I120_REJ_BIN_PRSNCE_I1221_0                    :BOOL;
I120_SPARE_I1221_1                             :BOOL;
I120_SPARE_I1221_2                             :BOOL;
I120_SPARE_I1221_3                             :BOOL;
I120_SPARE_I1221_4                             :BOOL;
I120_SPARE_I1221_5                             :BOOL;
I120_SPARE_I1221_6                             :BOOL;
I120_SPARE_I1221_7                             :BOOL;

//port 5
O90_RET_LH_GRIPR_CYL_CLSE_Q1240_0              :BOOL;
O90_RET_LH_GRIPR_CYL_OPN_Q1240_1               :BOOL;
O90_RET_RH_GRIPR_CYL_CLSE_Q1240_2              :BOOL;
O90_RET_RH_GRIPR_CYL_OPN_Q1240_3               :BOOL;
O90_POS_LOCK_CYL1_VLVE_1_Q1240_4               :BOOL;
O90_POS_LOCK_CYL1_VLVE_2_Q1240_5               :BOOL;
O90_POS_LOCK_CYL2_VLVE_1_Q1240_6               :BOOL;
O90_POS_LOCK_CYL2_VLVE_2_Q1240_7               :BOOL;
											  
O90_POSTN_SLIDE_CYL_REV_Q1241_0                :BOOL;
O90_POSTN_SLIDE_CYL_FWD_Q1241_1                :BOOL;
O90_LH_MOVR_SUP_VERT_CYL_DWN_Q1241_2           :BOOL;
O90_LH_MOVR_SUP_VERT_CYL_UP_Q1241_3            :BOOL;
O90_LH_MOVR_SUP_HORZ_CYL_REV_Q1241_4           :BOOL;
O90_LH_MOVR_SUP_HORZ_CYL_FWD_Q1241_5           :BOOL;
O90_RH_MOVR_SUP_VERT_CYL_DWN_Q1241_6           :BOOL;
O90_RH_MOVR_SUP_VERT_CYL_UP_Q1241_7            :BOOL;
											   
O90_RH_MOVR_SUP_HORZ_CYL_REV_Q1242_0           :BOOL;
O90_RH_MOVR_SUP_HORZ_CYL_FWD_Q1242_1           :BOOL;
O90_SPARE_Q1242_2                              :BOOL;
O90_SPARE_Q1242_3                              :BOOL;
O90_SPARE_Q1242_4                              :BOOL;
O90_SPARE_Q1242_5                              :BOOL;
O90_SPARE_Q1242_6                              :BOOL;
O90_SPARE_Q1242_7                              :BOOL;

//port6
O90_LH1_REJ_SLIDE_REV_Q1250_0                  :BOOL;
O90_LH1_REJ_SLIDE_FWD_Q1250_1                  :BOOL;
O90_RH1_REJ_SLIDE_REV_Q1250_2                  :BOOL;
O90_RH1_REJ_SLIDE_FWD_Q1250_3                  :BOOL;
O90_SPARE_Q1250_4                              :BOOL;
O90_LH1_REJ_AIR_PURGE_Q1250_5                  :BOOL;
O90_LH2_REJ_SLIDE_REV_Q1250_6                  :BOOL;
O90_LH2_REJ_SLIDE_FWD_Q1250_7                  :BOOL;
											  
O90_RH2_REJ_SLIDE_REV_Q1251_0                  :BOOL;
O90_RH2_REJ_SLIDE_FWD_Q1251_1                  :BOOL;
O90_RH_REJ_AIR_PURGE_Q1251_2                   :BOOL;
O90_SPARE_Q1251_3                              :BOOL;
O90_SPARE_Q1251_4                              :BOOL;
O90_SPARE_Q1251_5                              :BOOL;
O90_SPARE_Q1251_6                              :BOOL;
O90_SPARE_Q1251_7                              :BOOL;

//port7
O110_LH_OIL_DISPN_ON_Q1260_0                   :BOOL;
O110_LH_OIL_SPIN_ON_Q1260_1                    :BOOL;
O110_RH_OIL_DISPN_ON_Q1260_2                   :BOOL;
O110_RH_OIL_SPIN_ON_Q1260_3                    :BOOL;
O120_LH_GRPR_CLSE_Q1260_4                      :BOOL;
O120_LH_GRPR_OPN_Q1260_5                       :BOOL;
O120_RH_GRPR_CLSE_Q1260_6                      :BOOL;
O120_RH_GRPR_OPN_Q1260_7                       :BOOL;
											  
O120_TOOL_CHO_UNLOCK_Q1261_0                   :BOOL;
O120_TOOL_CHO_LOCK_Q1261_1                     :BOOL;
O120_PUSH_CYL_REV_Q1261_2                      :BOOL;
O120_PUSH_CYL_FWD_Q1261_3                      :BOOL;
O120_LH_SING_CYL_REV_Q1261_4                   :BOOL;
O120_LH_SING_CYL_FWD_Q1261_5                   :BOOL;
O120_LH_REJ_AIR_PURGE_Q1261_6                  :BOOL;
O120_RH_REJ_AIR_PURGE_Q1261_7                  :BOOL;
											  
O120_CAMERA_SLIDECYL_REV_Q1262_0               :BOOL;
O120_CAMERA_SLIDECYL_FWD_Q1262_1               :BOOL;
O120_SPARE_Q1262_2                             :BOOL;
O120_SPARE_Q1262_3                             :BOOL;
O120_SPARE_Q1262_4                             :BOOL;
O120_SPARE_Q1262_5                             :BOOL;
O120_SPARE_Q1262_6                             :BOOL;
O120_SPARE_Q1262_7                             :BOOL;
END_VAR

// ---- POUs/IO_GVLs/Master4_IO.TcGVL

VAR_GLOBAL
//port1					
I130_LH_ROTRY_0_DEGI1300_0                :BOOL;
I130_LH_ROTRY_180_DEGI1300_1              :BOOL;
I130_RH_ROTRY_0_DEGI1300_2                :BOOL;
I130_RH_ROTRY_180_DEGI1300_3              :BOOL;
I130_SPARE_I1300_4                        :BOOL;
I130_SPARE_I1300_5                        :BOOL;
I130_SPARE_I1300_6                        :BOOL;
I130_SPARE_I1300_7                        :BOOL;
										  
I140_HORZ_SUP1_CYL_REVI1301_0             :BOOL;
I140_HORZ_SUP1_CYL_FWDI1301_1             :BOOL;
I140_VERT_SUP1_CYL_REVI1301_2             :BOOL;
I140_VERT_SUP1_CYL_FWDI1301_3             :BOOL;
I140_WIPE1_CYL_REVI1301_4                 :BOOL;
I140_WIPE1_CYL_FWDI1301_5                 :BOOL;
I140_SPARE_I1301_6                        :BOOL;
I140_SPARE_I1301_7                        :BOOL;
										  
// port 2                         
I140_HORZ_SUP2_CYL_REVI1310_0             :BOOL;
I140_HORZ_SUP2_CYL_FWDI1310_1             :BOOL;
I140_VERT_SUP2_CYL_REVI1310_2             :BOOL;
I140_VERT_SUP2_CYL_FWDI1310_3             :BOOL;
I140_WIPE2_CYL_REVI1310_4                 :BOOL;
I140_WIPE2_CYL_FWDI1310_5                 :BOOL;
I140_HORZ_SUP3_CYL_REVI1310_6             :BOOL;
I140_HORZ_SUP3_CYL_FWDI1310_7             :BOOL;
										  
I140_VERT_SUP3_CYL_REVI1311_0             :BOOL;
I140_VERT_SUP3_CYL_FWDI1311_1             :BOOL;
I140_WIPE3_CYL_REVI1311_2                 :BOOL;
I140_WIPE3_CYL_FWDI1311_3                 :BOOL;
I140_LEAKTEST_PRESS_SWI1311_4             :BOOL;
I140_SPARE_I1311_5                        :BOOL;
I160_MOVR_REM_CYL_REVI1311_6             :BOOL;
I160_MOVR_REM_CYL_FWDI1311_7             :BOOL;
										  
// port 3                        									  
I160_SLIDE_CYL_REVI1320_0                 :BOOL;
I160_SLIDE_CYL_FWDI1320_1                 :BOOL;
I160_SLAVE1_PRSN_PARK_TRAYI1320_2         :BOOL;
I160_SLAVE2_PRSN_PARK_TRAYI1320_3         :BOOL;
I160_FIXT_COMP1_PRSNI1320_4               :BOOL;
I160_FIXT_COMP2_PRSNI1320_5               :BOOL;
I160_SPARE_I1320_6                        :BOOL;
I160_SPARE_I1320_7                        :BOOL;
										  
I160_SPARE_I1321_0                        :BOOL;
I160_SPARE_I1321_1                        :BOOL;
I160_SPARE_I1321_2                        :BOOL;
I160_SPARE_I1321_3                        :BOOL;
I160_SPARE_I1321_4                        :BOOL;
I160_SPARE_I1321_5                        :BOOL;
I160_SPARE_I1321_6                        :BOOL;
I160_SPARE_I1321_7                        :BOOL;
										  
// port 4                        
I160_LH_PALLET_LOCK_CYL_UNLOCKI1330_0     :BOOL;
I160_LH_PALLET_LOCK_CYL_LOCKI1330_1       :BOOL;
I160_RH_PALLET_LOCK_CYL_UNLOCKI1330_2     :BOOL;
I160_RH_PALLET_LOCK_CYL_LOCKI1330_3       :BOOL;
I160_SPARE_I1330_4                        :BOOL;
I160_CONV_BDY_PRSN1_SENI1330_5            :BOOL;
I160_CONV_BDY_PRSN2_SENI1330_6            :BOOL;
I160_SPARE_I1330_7                        :BOOL;
										  
I160_REJ_BOX_DOOR_CLSEI1331_0             :BOOL;
I160_SAM_PART_BAG_DOOR_CLSEI1331_1        :BOOL;
I160_TROLLEY_FIXT_PRSNI1331_2             :BOOL;
I160_SAM_BOX_DOOR_CLSEI1331_3             :BOOL;
I160_SPARE_I1331_4                        :BOOL;
I160_SPARE_I1331_5                        :BOOL;
I160_SPARE_I1331_6                        :BOOL;
I160_SPARE_I1331_7                        :BOOL;
										 
//PORT5                            									 
O130_LH_ROTRY_0_DEG_Q1340_0               :BOOL;
O130_LH_ROTRY_180_DEG_Q1340_1             :BOOL;
O130_RH_ROTRY_0_DEG_Q1340_2               :BOOL;
O130_RH_ROTRY_180_DEG_Q1340_3             :BOOL;
O130_LH_TOOL_CHO_UNLOCK_Q1340_4           :BOOL;
O130_LH_TOOL_CHO_LOCK_Q1340_5             :BOOL;
O130_RH_TOOL_CHO_UNLOCK_Q1340_6           :BOOL;
O130_RH_TOOL_CHO_LOCK_Q1340_7             :BOOL;
										 
O140_HORZ_SUP1_CYL_REV_Q1341_0            :BOOL;
O140_HORZ_SUP1_CYL_FWD_Q1341_1            :BOOL;
O140_VERT_SUP1_CYL_REV_Q1341_2            :BOOL;
O140_VERT_SUP1_CYL_FWD_Q1341_3            :BOOL;
O140_TOOL1_CHO_UNLOCK_Q1341_4             :BOOL;
O140_TOOL1_CHO_LOCK_Q1341_5               :BOOL;
O140_WIPE1_CYL_REV_Q1341_6                :BOOL;
O140_WIPE1_CYL_FWD_Q1341_7                :BOOL;
										  
O140_HORZ_SUP2_CYL_REV_Q1342_0            :BOOL;
O140_HORZ_SUP2_CYL_FWD_Q1342_1            :BOOL;
O140_VERT_SUP2_CYL_REV_Q1342_2            :BOOL;
O140_VERT_SUP2_CYL_FWD_Q1342_3            :BOOL;
O140_TOOL2_CHO_UNLOCK_Q1342_4             :BOOL;
O140_TOOL2_CHO_LOCK_Q1342_5               :BOOL;
O140_WIPE2_CYL_REV_Q1342_6                :BOOL;
O140_WIPE2_CYL_FWD_Q1342_7                :BOOL;
										  
O140_HORZ_SUP3_CYL_REV_Q1343_0            :BOOL;
O140_HORZ_SUP3_CYL_FWD_Q1343_1            :BOOL;
O140_VERT_SUP3_CYL_REV_Q1343_2            :BOOL;
O140_VERT_SUP3_CYL_FWD_Q1343_3            :BOOL;
O140_TOOL3_CHO_UNLOCK_Q1343_4             :BOOL;
O140_TOOL3_CHO_LOCK_Q1343_5               :BOOL;
O140_WIPE3_CYL_REV_Q1343_6                :BOOL;
O140_WIPE3_CYL_FWD_Q1343_7                :BOOL;
										  
//PORT6                           									  
O160_VISN_CHECK_AIR_PURGE_Q1350_0         :BOOL;
O160_FIXT_PP_GRPR_CLSE_OPN_Q1350_1        :BOOL;
O160_LH_COMP_PP_GRPR_CLSE_OPN_Q1350_2     :BOOL;
O160_RH_COMP_PP_GRPR_CLSE_OPN_Q1350_3     :BOOL;
O160_SLIDE_CYL_REV_Q1350_4                :BOOL;
O160_SLIDE_CYL_FWD_Q1350_5                :BOOL;
O160_SPARE_Q1350_6                        :BOOL;
O160_SPARE_Q1350_7                        :BOOL;
										 
O160_TOOL_CHO_UNLOCK_Q1351_0              :BOOL;
O160_TOOL_CHO_LOCK_Q1351_1                :BOOL;
O160_LH_PALLET_LOCK_CYL_UNLOCK_Q1351_2    :BOOL;
O160_LH_PALLET_LOCK_CYL_LOCK_Q1351_3      :BOOL;
O160_RH_PALLET_LOCK_CYL_UNLOCK_Q1351_4    :BOOL;
O160_RH_PALLET_LOCK_CYL_LOCK_Q1351_5      :BOOL;
O160_SPARE_Q1351_6                        :BOOL;
O160_SPARE_Q1351_7                        :BOOL;
										  
O160_SPARE_Q1352_0                        :BOOL;
O160_SPARE_Q1352_1                        :BOOL;
OP160_MOVR_REM_CYL_REV_Q1352_2           :BOOL;
OP160_MOVR_REM_CYL_FWD_Q1352_3           :BOOL;
O160_SPARE_Q1352_4                        :BOOL;
O160_SPARE_Q1352_5                        :BOOL;
O160_SPARE_Q1352_6                        :BOOL;
O160_SPARE_Q1352_7                        :BOOL;
										 
O160_SPARE_Q1353_0                        :BOOL;
O160_SPARE_Q1353_1                        :BOOL;
O160_SPARE_Q1353_2                        :BOOL;
O160_SPARE_Q1353_3                        :BOOL;
O160_SPARE_Q1353_4                        :BOOL;
O160_SPARE_Q1353_5                        :BOOL;
O160_SPARE_Q1353_6                        :BOOL;
O160_SPARE_Q1353_7                        :BOOL;
END_VAR

// ---- POUs/IO_GVLs/OP120_JB.TcGVL

VAR_GLOBAL

I120_SPARE_600_0I600_0             :BOOL;
I120_HPR_LOW_LVL_FBI600_1          :BOOL;
I120_HPR_SOL_DOOR_SW_FBI600_2      :BOOL;
I120_BOWL_RDYI600_3                :BOOL;
I120_BOWL_LOW_LVLI600_4            :BOOL;
I120_BOWL_OFF_ONI600_5             :BOOL;
I120_HPR_OFF_ONI600_6              :BOOL;
I120_CONV_REVI600_7                :BOOL;
I120_CONV_FWDI601_0                :BOOL;
I120_VBF_CONV_TRK1_OVERFLW_I601_1  :BOOL;
I120_VBF_CONV_TRK2_OVERFLWI601_2   :BOOL;
I120_CONV_TRK1_CHO_MOD1I601_3      :BOOL;
I120_CONV_TRK1_CHO_MOD2I601_4      :BOOL;
I120_CONV_TRK2_CHO_MOD1I601_5      :BOOL;
I120_CONV_TRK2_CHO_MOD2I601_6      :BOOL;
I120_CONV_TRK3_CHO_MOD1I601_7      :BOOL;
								   			   
I120_CONV_TRK3_CHO_MOD2I602_0      :BOOL;
I120_VBF_CONV_TRK_OVERFLW2_I602_1  :BOOL;
I120_SPARE_I602_2                  :BOOL;
I120_SPARE_I602_3                  :BOOL;
I120_SPARE_I602_4                  :BOOL;
I120_SPARE_I602_5                  :BOOL;
I120_SPARE_I602_6                  :BOOL;
I120_SPARE_I602_7                  :BOOL;
I120_SPARE_I603_0                  :BOOL;
I120_SPARE_I603_1                  :BOOL;
I120_SPARE_I603_2                  :BOOL;
I120_SPARE_I603_3                  :BOOL;
I120_SPARE_I603_4                  :BOOL;
I120_SPARE_I603_5                  :BOOL;
I120_SPARE_I603_6                  :BOOL;
I120_SPARE_I603_7                  :BOOL;

O120_HPR_ENABLEQ600_0              :BOOL;
O120_BOWL_ENABLEQ600_1             :BOOL;
O120_HPR_TWR_LMP_REDQ600_2         :BOOL;
O120_HPR_TWR_LMP_GREENQ600_3       :BOOL;
O120_BOWL_AIR_PURGE1Q600_4         :BOOL;
O120_BOWL_AIR_PURGE2Q600_5         :BOOL;
O120_HPR_DOOR_OPNQ600_6            :BOOL;
O120_SPARE_Q600_7                  :BOOL;
O120_SPARE_Q601_0                  :BOOL;
O120_SPARE_Q601_1                  :BOOL;
O120_SPARE_Q601_2                  :BOOL;
O120_SPARE_Q601_3                  :BOOL;
O120_SPARE_Q601_4                  :BOOL;
O120_SPARE_Q601_5                  :BOOL;
O120_SPARE_Q601_6                  :BOOL;
O120_SPARE_Q601_7                  :BOOL;

O120_SPARE_Q602_0                  :BOOL;
O120_SPARE_Q602_1                  :BOOL;
O120_SPARE_Q602_2                  :BOOL;
O120_SPARE_Q602_3                  :BOOL;
O120_SPARE_Q602_4                  :BOOL;
O120_SPARE_Q602_5                  :BOOL;
O120_SPARE_Q602_6                  :BOOL;
O120_SPARE_Q602_7                  :BOOL;
O120_SPARE_Q603_0                  :BOOL;
O120_SPARE_Q603_1                  :BOOL;
O120_SPARE_Q603_2                  :BOOL;
O120_SPARE_Q603_3                  :BOOL;
O120_SPARE_Q603_4                  :BOOL;
O120_SPARE_Q603_5                  :BOOL;
O120_SPARE_Q603_6                  :BOOL;
O120_SPARE_Q603_7                  :BOOL;
	
END_VAR

// ---- POUs/IO_GVLs/OP160_MP.TcGVL

VAR_GLOBAL
I130_LH_ATC_DECLAMP_FBI700_0				:BOOL;
I130_LH_ATC_CLAMP_FBI700_1                 :BOOL;
I130_LH_ATC_STN_POKE_YOKE_1I700_2          :BOOL;
I130_LH_ATC_STN_POKE_YOKE_2I700_3          :BOOL;
I130_LH_ATC_STN_POKE_YOKE_3I700_4          :BOOL;
I130_LH_ATC_STN_POKE_YOKE_4I700_5          :BOOL;
I130_LH_ATC_SLAVE_MODL1I700_6              :BOOL;
I130_LH_ATC_SLAVE_MODL2I700_7              :BOOL;
I130_RH_ATC_DECLAMP_FBI701_0               :BOOL;
I130_RH_ATC_CLAMP_FBI701_1                 :BOOL;
I130_RH_ATC_STN_POKE_YOKE_1I701_2          :BOOL;
I130_RH_ATC_STN_POKE_YOKE_2I701_3          :BOOL;
I130_RH_ATC_STN_POKE_YOKE_3I701_4          :BOOL;
I130_RH_ATC_STN_POKE_YOKE_4I701_5          :BOOL;
I130_RH_ATC_SLAVE_MODL1I701_6              :BOOL;
I130_RH_ATC_SLAVE_MODL2I701_7              :BOOL;

I140_ATC1_DECLAMP_FBI702_0                 :BOOL;
I140_ATC1_CLAMP_FBI702_1                   :BOOL;
I140_ATC1_STN_POKE_YOKE_1I702_2            :BOOL;
I140_ATC1_STN_POKE_YOKE_2I702_3            :BOOL;
I140_ATC1_STN_POKE_YOKE_3I702_4            :BOOL;
I140_ATC1_STN_POKE_YOKE_4I702_5            :BOOL;
I140_ATC1_SLAVE_MODL1I702_6                :BOOL;
I140_ATC1_SLAVE_MODL2I702_7                :BOOL;
I140_SPARE_I703_0                          :BOOL;
I140_SPARE_I703_1                          :BOOL;
I140_SPARE_I703_2                          :BOOL;
I140_LK_TST_1_PASI703_3                    :BOOL;
I140_LK_TST_1_FLI703_4                     :BOOL;
I140_LK_TST_1_REF_PRT_FLI703_5             :BOOL;
I140_LK_TST_1_WARNGI703_6                  :BOOL;
I140_LK_TST_1_END_CYCI703_7                :BOOL;

										  
I140_SPARE_I704_0I704_0                    :BOOL;
I140_LK_TST_2_PASI704_1                    :BOOL;
I140_LK_TST_2_FLI704_2                     :BOOL;
I140_LK_TST_2_REF_PRT_FLI704_3             :BOOL;
I140_LK_TST_2_WARNGI704_4                  :BOOL;
I140_LK_TST_2_END_CYCI704_5                :BOOL;
I140_SPARE_I704_6                          :BOOL;
I140_SPARE_I704_7                          :BOOL;
I140_ATC2_DECLAMP_FBI705_0                 :BOOL;
I140_ATC2_CLAMP_FBI705_1                   :BOOL;
I140_ATC2_STN_POKE_YOKE_1I705_2            :BOOL;
I140_ATC2_STN_POKE_YOKE_2I705_3            :BOOL;
I140_ATC2_STN_POKE_YOKE_3I705_4            :BOOL;
I140_ATC2_STN_POKE_YOKE_4I705_5            :BOOL;
I140_ATC2_SLAVE_MODL1I705_6                :BOOL;
I140_ATC2_SLAVE_MODL2I705_7                :BOOL;
										   

I140_SPARE_I706_0                          :BOOL;
I140_LK_TST_3_PASI706_1                    :BOOL;
I140_LK_TST_3_FLI706_2                     :BOOL;
I140_LK_TST_3_REF_PRT_FLI706_3             :BOOL;
I140_LK_TST_3_WARNGI706_4                  :BOOL;
I140_LK_TST_3_END_CYCI706_5                :BOOL;
I140_SPARE_I706_6                          :BOOL;
I140_SPARE_I706_7                          :BOOL;
I140_SPARE_I707_0                          :BOOL;
I140_LK_TST_4_PASI707_1                    :BOOL;
I140_LK_TST_4_FLI707_2                     :BOOL;
I140_LK_TST_4_REF_PRT_FLI707_3             :BOOL;
I140_LK_TST_4_WARNGI707_4                  :BOOL;
I140_LK_TST_4_END_CYCI707_5                :BOOL;
I140_SPARE_I707_6                          :BOOL;
I140_SPARE_I707_7                          :BOOL;


I140_ATC3_DECLAMP_FBI708_0                 :BOOL;
I140_ATC3_CLAMP_FBI708_1                   :BOOL;
I140_ATC3_STN_POKE_YOKE_1I708_2            :BOOL;
I140_ATC3_STN_POKE_YOKE_2I708_3            :BOOL;
I140_ATC3_STN_POKE_YOKE_3I708_4            :BOOL;
I140_ATC3_STN_POKE_YOKE_4I708_5            :BOOL;
I140_ATC3_SLAVE_MODL1I708_6                :BOOL;
I140_ATC3_SLAVE_MODL2I708_7                :BOOL;
I140_SPARE_I709_0                          :BOOL;
I140_SPARE_I709_1                          :BOOL;
I140_SPARE_I709_2                          :BOOL;
I140_LK_TST_5_PASI709_3                    :BOOL;
I140_LK_TST_5_FLI709_4                     :BOOL;
I140_LK_TST_5_REF_PRT_FLI709_5             :BOOL;
I140_LK_TST_5_WARNGI709_6                  :BOOL;
I140_LK_TST_5_END_CYCI709_7                :BOOL;

I140_SPARE_I710_0                          :BOOL;
I140_LK_TST_6_PASI710_1                    :BOOL;
I140_LK_TST_6_FLI710_2                     :BOOL;
I140_LK_TST_6_REF_PRT_FLI710_3             :BOOL;
I140_LK_TST_6_WARNGI710_4                  :BOOL;
I140_LK_TST_6_END_CYCI710_5                :BOOL;
I160_ATC_DECLAMP_FBI710_6                  :BOOL;
I160_ATC_CLAMP_FBI710_7                    :BOOL;
I160_ATC1_STN_POKE_YOKE_1I711_0            :BOOL;
I160_ATC1_STN_POKE_YOKE_2I711_1            :BOOL;
I160_ATC1_STN_POKE_YOKE_3I711_2            :BOOL;
I160_ATC1_STN_POKE_YOKE_4I711_3            :BOOL;
I160_ATC1_SLAVE_TOOL1I711_4                :BOOL;
I160_ATC1_SLAVE_TOOL2I711_5                :BOOL;
I160_FIXT_LH_COMP_PP_GRPR_CLSEI711_6       :BOOL;
I160_FIXT_LH_COMP_PP_GRPR_OPNI711_7        :BOOL;
I160_RH_COMP_PP_GRPR_CLSEI712_0            :BOOL;
I160_RH_COMP_PP_GRPR_OPNI712_1             :BOOL;
I160_AUTOBAG_READYI712_2                   :BOOL;
I160_SPARE_I712_3                          :BOOL;
I160_SPARE_I712_4                          :BOOL;
I160_AUTOBAG_ERR_STOPI712_5                :BOOL;
I20_RESRVR_LW_LVLI712_6                    :BOOL;
I20_OILTANK_PRES_SW_FBI712_7               :BOOL;
I160_SPARE_I713_0                          :BOOL;
I160_SPARE_I713_1                          :BOOL;
I160_VFD_RDYI713_2                         :BOOL;
I160_SPARE_I713_3                          :BOOL;
I160_SPARE_I713_4                          :BOOL;
I160_SPARE_I713_5                          :BOOL;
I160_SPARE_I713_6                          :BOOL;
I160_SPARE_I713_7                          :BOOL;


I10A_DRUM_FEED_ALRMI714_0                  :BOOL;
I10A_SPARE_I714_1                          :BOOL;
I10A_DRUM_OFF_ON_I714_2                    :BOOL;
I10A_DRUM_CONV_REV_I714_3                  :BOOL;
I10A_DRUM_CONV_FWD_I714_4                  :BOOL;
I10A_ROB_MAN_AUTO_MODE_I714_5              :BOOL;
I160_SPARE_I714_6                          :BOOL;
I160_SPARE_I714_7                          :BOOL;
I160_SPARE_I715_0                          :BOOL;
I160_SPARE_I715_1                          :BOOL;
I160_SPARE_I715_2                          :BOOL;
I160_SPARE_I715_3                          :BOOL;
I160_SPARE_I715_4                          :BOOL;
I160_SPARE_I715_5                          :BOOL;
I160_SPARE_I715_6                          :BOOL;
I160_SPARE_I715_7                          :BOOL;

O140_LK_TST1_RST_Q700_0                   :BOOL;
O140_LK_TST1_STRT_Q700_1                  :BOOL;
O140_LK_TST1_SEL1_Q700_2                  :BOOL;
O140_LK_TST1_SEL2_Q700_3                  :BOOL;
O140_LK_TST1_SEL3_Q700_4                  :BOOL;
O140_LK_TST1_SEL4_Q700_5                  :BOOL;
O140_LK_TST1_SEL5_Q700_6                  :BOOL;
O140_LK_TST1_SEL6_Q700_7                  :BOOL;
O140_LK_TST1_SEL7_Q701_0                  :BOOL;
O140_LK_TST2_RST_Q701_1                   :BOOL;
O140_LK_TST2_STRT_Q701_2                  :BOOL;
O140_LK_TST2_SEL1_Q701_3                  :BOOL;
O140_LK_TST2_SEL2_Q701_4                  :BOOL;
O140_LK_TST2_SEL3_Q701_5                  :BOOL;
O140_LK_TST2_SEL4_Q701_6                  :BOOL;
O140_LK_TST2_SEL5_Q701_7                  :BOOL;

O140_LK_TST2_SEL6_Q702_0                  :BOOL;
O140_LK_TST2_SEL7_Q702_1                  :BOOL;
O140_LK_TST3_RST_Q702_2                   :BOOL;
O140_LK_TST3_STRT_Q702_3                  :BOOL;
O140_LK_TST3_SEL1_Q702_4                  :BOOL;
O140_LK_TST3_SEL2_Q702_5                  :BOOL;
O140_LK_TST3_SEL3_Q702_6                  :BOOL;
O140_LK_TST3_SEL4_Q702_7                  :BOOL;
O140_LK_TST3_SEL5_Q703_0                  :BOOL;
O140_LK_TST3_SEL6_Q703_1                  :BOOL;
O140_LK_TST3_SEL7_Q703_2                  :BOOL;
O140_LK_TST4_RST_Q703_3                   :BOOL;
O140_LK_TST4_STRT_Q703_4                  :BOOL;
O140_LK_TST4_SEL1_Q703_5                  :BOOL;
O140_LK_TST4_SEL2_Q703_6                  :BOOL;
O140_LK_TST4_SEL3_Q703_7                  :BOOL;

O140_LK_TST4_SEL4_Q704_0                  :BOOL;
O140_LK_TST4_SEL5_Q704_1                  :BOOL;
O140_LK_TST4_SEL6_Q704_2                  :BOOL;
O140_LK_TST4_SEL7_Q704_3                  :BOOL;
O140_LK_TST5_RST_Q704_4                   :BOOL;
O140_LK_TST5_STRT_Q704_5                  :BOOL;
O140_LK_TST5_SEL1_Q704_6                  :BOOL;
O140_LK_TST5_SEL2_Q704_7                  :BOOL;
O140_LK_TST5_SEL3_Q705_0                  :BOOL;
O140_LK_TST5_SEL4_Q705_1                  :BOOL;
O140_LK_TST5_SEL5_Q705_2                  :BOOL;
O140_LK_TST5_SEL6_Q705_3                  :BOOL;
O140_LK_TST5_SEL7_Q705_4                  :BOOL;
O140_LK_TST6_RST_Q705_5                   :BOOL;
O140_LK_TST6_STRT_Q705_6                  :BOOL;
O140_LK_TST6_SEL1_Q705_7                  :BOOL;
										   

O140_LK_TST6_SEL2_Q706_0                  :BOOL;
O140_LK_TST6_SEL3_Q706_1                  :BOOL;
O140_LK_TST6_SEL4_Q706_2                  :BOOL;
O140_LK_TST6_SEL5_Q706_3                  :BOOL;
O140_LK_TST6_SEL6_Q706_4                  :BOOL;
O140_LK_TST6_SEL7_Q706_5                  :BOOL;
O150_VISN_LGHT_ON_Q706_6                   :BOOL;
O150_BARLIGHT_OP1_Q706_7                   :BOOL;
O150_BARLIGHT_OP2_Q707_0                   :BOOL;
O160_CHECKER_LGHT_ON_Q707_1                :BOOL;
O160_FUME_EXTRTR_ON_Q707_2                 :BOOL;
O160_MC_LMP_ON_Q707_3                      :BOOL;
O160_AUTOBAG_CNT_CMPLTD_Q707_4             :BOOL;
O160_SAMPLE_PART_DOOR_OPN_Q707_5           :BOOL;
O160_REJ_BIN_DOOR_OPN_Q707_6               :BOOL;
O160_SPARE_Q707_7                          :BOOL;
										   
O160_VFD_FWD_Q708_0                        :BOOL;
O160_VFD_REV_Q708_1                        :BOOL;
O160_VFD_STOP_Q708_2                       :BOOL;
O160_BOT_MC_LMP_ON_Q708_3                  :BOOL;
O10A_DRUM_MTR_FWD_Q708_4                   :BOOL;
O10A_DRUM_RST_Q708_5                       :BOOL;
O10A_DRUM_EXT_SPEED_Q708_6                 :BOOL;
O160_SPARE_Q708_7                          :BOOL;
O10A_DRUM_RUN_IND_Q709_0                   :BOOL;
O160_SPARE_Q709_1_Q709_1                   :BOOL;
O10A_ROB_MAN_AUTO_MODE_Q709_2              :BOOL;
O10B_ROB_MAN_AUTO_MODE_Q709_3              :BOOL;
O120_ROB_MAN_AUTO_MODE_Q709_4              :BOOL;
O160_SPARE_Q709_5                          :BOOL;
O160_SPARE_Q709_6                          :BOOL;
O160_SPARE_Q709_7                          :BOOL;
END_VAR

// ---- POUs/IO_GVLs/OP90_JB.TcGVL

VAR_GLOBAL
I90_SPARE_I500_0                     :BOOL;
I90_HPR1_LOW_LVL_FBI500_1            :BOOL;
I90_HPR1_SOL_DOOR_SW_FBI500_2        :BOOL;
I90_BOWL1_RDYI500_3                  :BOOL;
I90_BOWL1_LOW_LVLI500_4              :BOOL;
I90_BOWL1_OFF_ONI500_5               :BOOL;
I90_HPR1_OFF_ONI500_6                :BOOL;
I90_CONV1_REVI500_7                  :BOOL;
I90_CONV1_FWDI501_0                  :BOOL;
I90_VBF1_CONV1_TRK1_OVERFLWI501_1    :BOOL;
I90_VBF1_CONV1_TRK2_OVERFLWI501_2    :BOOL;
I90_CONV1_TRK1_CHO_MOD1I501_3        :BOOL;
I90_CONV1_TRK1_CHO_MOD2I501_4        :BOOL;
I90_CONV1_TRK2_CHO_MOD1I501_5        :BOOL;
I90_CONV1_TRK2_CHO_MOD2I501_6        :BOOL;
I90_CONV1_TRK3_CHO_MOD1I501_7        :BOOL;


I90_CONV1_TRK3_CHO_MOD2I502_0        :BOOL;
I90_SPARE_I502_1                     :BOOL;
I90_HPR2_LOW_LVL_FBI502_2            :BOOL;
I90_HPR2_SOL_DOOR_SW_FBI502_3        :BOOL;
I90_BOWL2_RDYI502_4                  :BOOL;
I90_BOWL2_LOW_LVLI502_5              :BOOL;
I90_BOWL2_OFF_ONI502_6               :BOOL;
I90_HPR2_OFF_ONI502_7                :BOOL;
I90_CONV2_REVI503_0                  :BOOL;
I90_CONV2_FWDI503_1                  :BOOL;
I90_VBF1_CONV2_TRK1_OVERFLWI503_2    :BOOL;
I90_VBF1_CONV2_TRK2_OVERFLWI503_3    :BOOL;
I90_CONV2_TRK1_CHO_MOD1I503_4        :BOOL;
I90_CONV2_TRK1_CHO_MOD2I503_5        :BOOL;
I90_CONV2_TRK2_CHO_MOD1I503_6        :BOOL;
I90_CONV2_TRK2_CHO_MOD2I503_7        :BOOL;


I90_CONV2_TRK3_CHO_MOD1I504_0        :BOOL;
I90_CONV2_TRK3_CHO_MOD2I504_1        :BOOL;
I90_VBF1_CONV_TRK_OVERFLW_2I504_2    :BOOL;
I90_VBF2_CONV_TRK_OVERFLW_2I504_3    :BOOL;
I90_SPARE_I504_4                     :BOOL;
I90_SPARE_I504_5                     :BOOL;
I90_SPARE_I504_6                     :BOOL;
I90_SPARE_I504_7                     :BOOL;
I90_SPARE_I505_0                     :BOOL;
I90_SPARE_I505_1                     :BOOL;
I90_SPARE_I505_2                     :BOOL;
I90_SPARE_I505_3                     :BOOL;
I90_SPARE_I505_4                     :BOOL;
I90_SPARE_I505_5                     :BOOL;
I90_SPARE_I505_6                     :BOOL;
I90_SPARE_I505_7                     :BOOL;


O90_HPR1_ENABLEQ500_0                :BOOL;
O90_BOWL1_ENABLEQ500_1               :BOOL;
O90_HPR1_TWR_LMP_REDQ500_2           :BOOL;
O90_HPR1_TWR_LMP_GREENQ500_3         :BOOL;
O90_BOWL1_AIR_PURGE1Q500_4           :BOOL;
O90_BOWL1_AIR_PURGE2Q500_5           :BOOL;
O90_HPR1_DOOR_OPNQ500_6              :BOOL;
O90_SPARE_Q500_7                     :BOOL;
O90_HPR2_ENABLEQ501_0                :BOOL;
O90_BOWL2_ENABLEQ501_1               :BOOL;
O90_HPR2_TWR_LMP_REDQ501_2           :BOOL;
O90_HPR2_TWR_LMP_GREENQ501_3         :BOOL;
O90_BOWL2_AIR_PURGE1Q501_4           :BOOL;
O90_BOWL2_AIR_PURGE2Q501_5           :BOOL;
O90_HPR2_DOOR_OPNQ501_6              :BOOL;
O90_SPARE_Q501_7                     :BOOL;


O90_SPARE_Q502_0                     :BOOL;
O90_SPARE_Q502_1                     :BOOL;
O90_SPARE_Q502_2                     :BOOL;
O90_SPARE_Q502_3                     :BOOL;
O90_SPARE_Q502_4                     :BOOL;
O90_SPARE_Q502_5                     :BOOL;
O90_SPARE_Q502_6                     :BOOL;
O90_SPARE_Q502_7                     :BOOL;
O90_SPARE_Q503_0                     :BOOL;
O90_SPARE_Q503_1                     :BOOL;
O90_SPARE_Q503_2                     :BOOL;
O90_SPARE_Q503_3                     :BOOL;
O90_SPARE_Q503_4                     :BOOL;
O90_SPARE_Q503_5                     :BOOL;
O90_SPARE_Q503_6                     :BOOL;
O90_SPARE_Q503_7                     :BOOL;

END_VAR

// ---- POUs/IO_GVLs/OP90_MP.TcGVL

VAR_GLOBAL
I90_PMR_FB_I400_0				:BOOL;
I90_SURGE_ARRES_FB_I400_1       :BOOL;
I90_DOOR1_CLOSE_FB_I400_2       :BOOL;
I90_DOOR2_CLOSE_FB_I400_3       :BOOL;
I90_DOOR3_CLOSE_FB_I400_4       :BOOL;
I90_DOOR4_CLOSE_FB_I400_5       :BOOL;
I90_DOOR5_CLOSE_FB_I400_6       :BOOL;
I90_DOOR6_CLOSE_FB_I400_7       :BOOL;
I90_DOOR7_CLOSE_FB_I401_0       :BOOL;
I90_DOOR8_CLOSE_FB_I401_1       :BOOL;
I90_DOOR9_CLOSE_FB_I401_2       :BOOL;
I90_DOOR10_CLOSE_FB_I401_3      :BOOL;
I90_DOOR11_CLOSE_FB_I401_4      :BOOL;
I90_DOOR12_CLOSE_FB_I401_5      :BOOL;
I90_DOOR13_CLOSE_FB_I401_6      :BOOL;
I90_DOOR14_CLOSE_FB_I401_7      :BOOL;

I90_DOOR15_CLOSE_FB_I402_0      :BOOL;
I90_DOOR16_CLOSE_FB_I402_1      :BOOL;
I110_RESRVR_LW_LVL_I402_2       :BOOL;
I110_OILTANK_PRES_SW_FB_I402_3  :BOOL;
I120_ATC_DECLAMP_FB_I402_4      :BOOL;
I120_ATC_CLAMP_FB_I402_5        :BOOL;
I120_ATC_STN_POKE_YOKE_1_I402_6 :BOOL;
I120_ATC_STN_POKE_YOKE_2_I402_7 :BOOL;
I120_ATC_STN_POKE_YOKE_3_I403_0 :BOOL;
I120_ATC_STN_POKE_YOKE_4_I403_1 :BOOL;
I120_ATC_SLAVE_MODL1_I403_2     :BOOL;
I120_ATC_SLAVE_MODL2_I403_3     :BOOL;
I120_SPARE_I403_4               :BOOL;
I120_SPARE_I403_5               :BOOL;
I120_SPARE_I403_6               :BOOL;
I90_RESET_FB_I403_7             :BOOL;

I90_LHS_ESTOP1_FB_I404_0        :BOOL;
I90_LHS_ESTOP2_FB_I404_1        :BOOL;
I90_LHS_ESTOP3_FB_I404_2        :BOOL;
I90_RHS_ESTOP1_FB_I404_3        :BOOL;
I90_RHS_ESTOP2_FB_I404_4        :BOOL;
I90_RHS_ESTOP3_FB_I404_5        :BOOL;
I90_SPARE_I404_6                :BOOL;
I90_SPARE_I404_7                :BOOL;
I90_XTS_48VSMPS1_DC_OK_I405_0   :BOOL;
I90_XTS_48VSMPS2_DC_OK_I405_1   :BOOL;
I90_XTS_48VSMPS3_DC_OK_I405_2   :BOOL;
I90_XTS_24VSMPS_DC_OK_I405_3    :BOOL;
I120_LH_LOCKSPRING_GRPR_CLSE_I405_4:BOOL;
I120_LH_LOCKSPRING_GRPR_OPN_I405_5 :BOOL;
I120_RH_LOCKSPRING_GRPR_CLSE_I405_6 :BOOL;
I120_RH_LOCKSPRING_GRPR_OPN_I405_7 :BOOL;

O90_VISN_LGHT1_ON_Q400_0        :BOOL;
O90_VISN_LGHT2_ON_Q400_1        :BOOL;
O90_LH_DOOR_OPN_Q400_2          :BOOL;
O90_RH_DOOR_OPN_Q400_3          :BOOL;
O90_FRNT_DOOR_OPN_Q400_4        :BOOL;
O90_BACK_DOOR_OPN_Q400_5        :BOOL;
O90_IPC_P_S_Q400_6              :BOOL;
O90_SPARE_Q400_7                :BOOL;
O90_SPARE_Q401_0                :BOOL;
O90_SPARE_Q401_1                :BOOL;
O90_SPARE_Q401_2                :BOOL;
O90_SPARE_Q401_3                :BOOL;
O110_RH_OIL_DISPN_FRL_VLVE_ON_Q401_4   :BOOL;
O20_RH_OIL_DISPN_FRL_VLVE_ON_Q401_5    :BOOL;
O110_LH_OIL_DISPN_FRL_VLVE_ON_Q401_6   :BOOL;
O20_LH_OIL_DISPN_FRL_VLVE_ON_Q401_7    :BOOL;

O110_SPARE_Q402_0               :BOOL;
O110_SPARE_Q402_1               :BOOL;
O110_SPARE_Q402_2               :BOOL;
O110_SPARE_Q402_3               :BOOL;
O120_VISN_LGHT1_ON_Q402_4       :BOOL;
O120_VISN_LGHT2_ON_Q402_5       :BOOL;
O120_BARLIGHT_OP1_Q402_6        :BOOL;
O120_BARLIGHT_OP2_Q402_7        :BOOL;
O120_TWR_LMP_RD_Q403_0          :BOOL;
O120_TWR_LMP_GN_Q403_1          :BOOL;
O120_TWR_LMP_YELW_Q403_2        :BOOL;
O120_TWR_LMP_BUZZ_Q403_3        :BOOL;
O120_SPARE_Q403_4               :BOOL;
O120_SPARE_Q403_5               :BOOL;
O120_SPARE_Q403_6               :BOOL;
O120_SPARE_Q403_7               :BOOL;	
END_VAR

// ---- POUs/IO_GVLs/SAFETY_IOs.TcGVL

VAR_GLOBAL
IS90_DOORSW_SET1_CH1_IS400_0 :BOOL;
IS90_DOORSW_SET2_CH1_IS400_1 :BOOL;
IS90_DOORSW_SET3_CH1_IS400_2 :BOOL;
IS90_DOORSW_SET4_CH1_IS400_3 :BOOL;
IS90_DOORSW_SET1_CH2_IS400_4 :BOOL;
IS90_DOORSW_SET2_CH2_IS400_5 :BOOL;
IS90_DOORSW_SET3_CH2_IS400_6 :BOOL;
IS90_DOORSW_SET4_CH2_IS400_7 :BOOL;
IS90_DOORSW_SET5_CH1_IS401_0 :BOOL;
IS90_DOORSW_SET6_CH1_IS401_1 :BOOL;
IS90_LHS_ESTOP_CH1_IS401_2   :BOOL;
IS90_RHS_ESTOP_CH1_IS401_3   :BOOL;
IS90_DOORSW_SET5_CH2_IS401_4 :BOOL;
IS90_DOORSW_SET6_CH2_IS401_5 :BOOL;
IS90_LHS_ESTOP_CH2_IS401_6   :BOOL;
IS90_RHS_ESTOP_CH2_IS401_7   :BOOL;
IS90_ESTOP_CONT_EDM_IS402_0  :BOOL;
IS90_DOOR_CONT_EDM_IS402_1   :BOOL;
IS90_RESET_IS402_2   :BOOL;
IS90_SPARE_IS402_3   :BOOL;
IS90_SPARE_IS402_4   :BOOL;
IS90_SPARE_IS402_5   :BOOL;
IS90_SPARE_IS402_6   :BOOL;
IS90_SPARE_IS402_7   :BOOL;
IS160_ESTOP_CONT_EDM_IS700_0 :BOOL;
IS160_DOOR_CONT_EDM_IS700_1  :BOOL;
IS160_SPARE_IS700_2  :BOOL;
IS160_SPARE_IS700_3  :BOOL;
IS160_SPARE_IS700_4  :BOOL;
IS160_SPARE_IS700_5  :BOOL;
IS160_SPARE_IS700_6  :BOOL;
IS160_SPARE_IS700_7  :BOOL;


OS90_ESTOP_CH1_QS400_0		:BOOL;
OS90_ESTOP_CH2_QS400_1      :BOOL;
OS90_DOORCH1_QS400_2        :BOOL;
OS90_DOORCH2_QS400_3        :BOOL;
OS160_ESTOP_CH1_QS700_0     :BOOL;
OS160_ESTOP_CH2_QS700_1     :BOOL;
OS160_DOORCH1_QS700_2       :BOOL;
OS160_DOORCH2_QS700_3       :BOOL;


END_VAR

// ---- POUs/IO_Mapping_OP10JB/IO_OP10_JB_IO.TcGVL

VAR_GLOBAL
	
	I10A_HPR_UNIT_ALRM_I100_0       :BOOL;
	I10A_SPARE_I100_1               :bool;
	I10A_HPR_LOW_LVL_SEN_I100_2     :bool;
	I10A_HPR_SOL_DOOR_SW_FB_I100_3  :bool;
	I10A_HPR_OFF_ON_I100_4          :bool;
	I10A_BDY_BOWL_OFF_ON_I100_5     :bool;
	I10A_BDY_LNR1_OFF_ON_I100_6     :bool;
	I10A_BDY_LNR2_OFF_ON_I100_7     :bool;
	I10A_HPR_DOOR_SELCTN_I101_0     :bool;
	I10A_SPARE_I101_1               :bool;
	I10A_BDY_BOWL_LOW_LVL_I101_2    :bool;
	I10A_BDY_BWL_RUN_I101_3         :bool;
	I10A_BDY_LNR1_RUN_I101_4        :bool;
	I10A_BDY_LNR2_RUN_I101_5        :bool;
	I10A_BDY_LNR_FEED1_OVRFLW_I101_6:bool;
	I10A_BDY_LNR_FEED2_OVRFLW_I101_7:bool;
	I10A_LNR_TRK1_CHO_MOD1_I102_0   :bool;
	I10A_LNR_TRK1_CHO_MOD2_I102_1   :bool;
	I10A_LNR_TRK2_CHO_MOD1_I102_2   :bool;
	I10A_LNR_TRK2_CHO_MOD2_I102_3   :bool;
	I10A_SPARE_I102_4               :BOOL;
	I10A_SPARE_I102_5               :BOOL;
	I10A_LH_BDY_CONT_FB_I102_6      :bool;
	I10A_RH_BDY_CONT_FB_I102_7      :bool;
	I10A_SPARE_I103_0               :bool;
	I10A_SPARE_I103_1               :bool;
	I10A_SPARE_I103_2               :bool;
	I10A_SPARE_I103_3               :bool;
	I10A_SPARE_I103_4               :bool;
	I10A_SPARE_I103_5               :bool;
	I10A_SPARE_I103_6               :bool;
	I10A_SPARE_I103_7               :BOOL;
	
	O10A_HPR_MTR_FWD_Q100_0        : BOOL;   
	O10A_HPR_RST_Q100_1            : BOOL;   
	O10A_EXT_SPEED_Q100_2          : Bool;   
	O10A_SPARE_Q100_3       		: BOOL;   
	O10A_HPR_DOOR_SELCTN_IND_Q100_4: Bool;   
	O10A_HPR_TWR_LMP_RED_Q100_5    : Bool;   
	O10A_HPR_TWR_LMP_GREEN_Q100_6  : Bool;   
	O10A_SPARE_Q100_7       	   : BOOL;   
	O10A_BDY_BOWL_ON_Q101_0        : Bool;   
	O10A_BDY_LNR_FEED1_ON_Q101_1   : Bool;   
	O10A_BDY_LNR_FEED2_ON_Q101_2   : Bool;   
	O10A_BDY_LNR1_AIR_PURGE_Q101_3 : Bool;   
	O10A_BDY_LNR2_AIR_PURGE_Q101_4 : Bool;   
	O10A_HPR_DOOR_OPN_Q101_5       : Bool;   
	O10A_SPARE_Q101_6              : Bool;   
	O10A_SPARE_Q101_7              : Bool;   
	O10A_SPARE_Q102_0              : Bool;   
	O10A_SPARE_Q102_1              : Bool;   
	O10A_SPARE_Q102_2              : Bool;   
	O10A_SPARE_Q102_3              : Bool;   
	O10A_SPARE_Q102_4              : Bool;   
	O10A_SPARE_Q102_5              : Bool;   
	O10A_SPARE_Q102_6              : Bool;   
	O10A_SPARE_Q102_7              : Bool;   
	O10A_SPARE_Q103_0              : Bool;   
	O10A_SPARE_Q103_1              : Bool;   
	O10A_SPARE_Q103_2              : Bool;   
	O10A_SPARE_Q103_3              : Bool;   
	O10A_SPARE_Q103_4              : Bool;   
	O10A_SPARE_Q103_5              : Bool;   
	O10A_SPARE_Q103_6              : Bool;   
	O10A_SPARE_Q103_7              : BOOL;

	I10B_HPR_UNIT_ALRM_I200_0          :BOOL;
	I10B_SPARE_I200_1                  :BOOL;
	I10B_HPR_LOW_LVL_SEN_I200_2        :BOOL;
	I10B_HPR_SOL_DOOR_SW_FB_I200_3     :BOOL;
	I10B_HPR_OFF_ON_I200_4             :BOOL;
	I10B_BDY_BOWL_OFF_ON_I200_5        :BOOL;
	I10B_BDY_LNR1_OFF_ON_I200_6        :BOOL;
	I10B_BDY_LNR2_OFF_ON_I200_7        :BOOL;
	I10B_HPR_DOOR_SELCTN_I201_0        :BOOL;
	I10B_SPARE_I201_1			       :BOOL;
	I10B_BDY_BOWL_LOW_LVL_I201_2       :BOOL;
	I10B_BDY_BWL_RUN_I201_3            :BOOL;
	I10B_BDY_LNR1_RUN_I201_4           :BOOL;
	I10B_BDY_LNR2_RUN_I201_5           :BOOL;
	I10B_BDY_LNR_FEED1_OVRFLW_I201_6   :BOOL;
	I10B_BDY_LNR_FEED2_OVRFLW_I201_7   :BOOL;
	I10B_LNR_TRK1_CHO_MOD1_I202_0      :BOOL;
	I10B_LNR_TRK1_CHO_MOD2_I202_1      :BOOL;
	I10B_LNR_TRK2_CHO_MOD1_I202_2      :BOOL;
	I10B_LNR_TRK2_CHO_MOD2_I202_3      :BOOL;
	I10B_SPARE_I202_4                  :BOOL;
	I10B_SPARE_I202_5     		       :BOOL;
	I10B_SPARE_I202_6           :BOOL;
	I10B_SPARE_I202_7           :BOOL;
	I10B_SPARE_I203_0           :BOOL;
	I10B_SPARE_I203_1           :BOOL;
	I10B_SPARE_I203_2           :BOOL;
	I10B_SPARE_I203_3           :BOOL;
	I10B_SPARE_I203_4           :BOOL;
	I10B_SPARE_I203_5           :BOOL;
	I10B_SPARE_I203_6           :BOOL;
	I10B_SPARE_I203_7		    :BOOL;
	
	O10B_HPR_MTR_FWD_Q200_0:BOOL;
	O10B_HPR_RST_Q200_1				 :BOOL;  
	O10B_EXT_SPEED_Q200_2            :bool;  
	O10B_SPARE_Q200_3		         :BOOL;  
	O10B_HPR_DOOR_SELCTN_IND_Q200_4  :bool;  
	O10B_HPR_TWR_LMP_RED_Q200_5      :bool;  
	O10B_HPR_TWR_LMP_GREEN_Q200_6    :bool;  
	O10B_SPARE_Q200_7                :BOOL;  
	O10B_BDY_BOWL_ON_Q201_0          :bool;  
	O10B_BDY_LNR_FEED1_ON_Q201_1     :bool;  
	O10B_BDY_LNR_FEED2_ON_Q201_2     :bool;  
	O10B_BDY_LNR1_AIR_PURGE_Q201_3   :bool;  
	O10B_BDY_LNR2_AIR_PURGE_Q201_4   :bool;  
	O10B_HPR_DOOR_OPN_Q201_5         :bool;  
	O10B_SPARE_Q201_6                :bool;  
	O10B_SPARE_Q201_7                :bool;  
	O10B_SPARE_Q202_0                :bool;  
	O10B_SPARE_Q202_1                :bool;  
	O10B_SPARE_Q202_2                :bool;  
	O10B_SPARE_Q202_3                :bool;  
	O10B_SPARE_Q202_4                :bool;  
	O10B_SPARE_Q202_5                :bool;  
	O10B_SPARE_Q202_6                :bool;  
	O10B_SPARE_Q202_7                :bool;  
	O10B_SPARE_Q203_0                :bool;  
	O10B_SPARE_Q203_1                :bool;  
	O10B_SPARE_Q203_2                :bool;  
	O10B_SPARE_Q203_3                :bool;  
	O10B_SPARE_Q203_4                :bool;  
	O10B_SPARE_Q203_5                :bool;  
	O10B_SPARE_Q203_6                :bool;  
	O10B_SPARE_Q203_7	             :BOOL;
END_VAR

// ---- POUs/IO_mapping_OP10MP/IO_OP10_MP.TcGVL

VAR_GLOBAL
		I10A_SPARE_I300_0						: BOOL;
		I10A_SPARE_I300_1                       : BOOL;
		I10A_SPARE_I300_2                       : BOOL;
		I10A_SPARE_I300_3                       : BOOL;
		I10A_SPARE_I300_4                       : BOOL;
		I10A_SPARE_I300_5                       : BOOL;
		I10A_SPARE_I300_6                       : BOOL;
		I10A_SPARE_I300_7                       : BOOL;
		I10A_SPARE_I301_0                       : BOOL;
		I10A_SPARE_I301_1                       : BOOL;
		I10A_SPARE_I301_2                       : BOOL;
		I10A_SPARE_I301_3                       : BOOL;
		I10A_SPARE_I301_4                       : BOOL;
		I10A_SPARE_I301_5                       : BOOL;
		I10A_SPARE_I301_6                       : BOOL;
		I10A_SPARE_I301_7                       : BOOL;
		
		I10B_DRUM_FEED_ALRM_I302_0              : BOOL;
		I10A_SPARE_I302_1                       : BOOL;
		I10B_DRUM_OFF_ON_I302_2                 : BOOL;
		I10B_DRUM_CONV_REV_I302_3               : BOOL;
		I10B_DRUM_CONV_FWD_I302_4               : BOOL;
		I10B_ROB_MAN_AUTO_MODE_I302_5           : BOOL;
		I10B_SPARE_I302_6                       : BOOL;
		I10B_SPARE_I302_7                       : BOOL;
		I10B_SPARE_I303_0                       : BOOL;
		I10B_SPARE_I303_1                       : BOOL;
		I10B_SPARE_I303_2                       : BOOL;
		I10B_SPARE_I303_3                       : BOOL;
		I10B_SPARE_I303_4                       : BOOL;
		I10B_SPARE_I303_5                       : BOOL;
		I10B_SPARE_I303_6                       : BOOL;
		I10B_SPARE_I303_7                       : BOOL;
		
		I30_DRUM_FEED_ALRM_I304_0               : BOOL;
		I30_SPARE_I304_1                        : BOOL;
		I30_DRUM_OFF_ON_I304_2                  : BOOL;
		I30_DRUM_CONV_REV_I304_3                : BOOL;
		I30_DRUM_CONV_FWD_I304_4                : BOOL;
		I30_SPARE_I304_5                        : BOOL;
		I30_SPARE_I304_6                        : BOOL;
		I30_SPARE_I304_7                        : BOOL;
		I40_ATC_DECLAMP_FB_I305_0               : BOOL;
		I40_ATC_CLAMP_FB_I305_1                 : BOOL;
		I40_ATC_STN_POKE_YOKE_1_I305_2          : BOOL;
		I40_ATC_STN_POKE_YOKE_2_I305_3          : BOOL;
		I40_ATC_STN_POKE_YOKE_3_I305_4          : BOOL;
		I40_ATC_STN_POKE_YOKE_4_I305_5          : BOOL;
		I40_ATC_SLAVE_MODL1_I305_6              : BOOL;
		I40_ATC_SLAVE_MODL2_I305_7              : BOOL;
		
		I50_DRUM_FEED_ALRM_I306_0               : BOOL;
		I50_SPARE_I306_1                        : BOOL;
		I50_DRUM_OFF_ON_I306_2                  : BOOL;
		I50_DRUM_CONV_REV_I306_3                : BOOL;
		I50_DRUM_CONV_FWD_I306_4                : BOOL;
		I50_SPARE_I306_5                        : BOOL;
		I50_SPARE_I306_6                        : BOOL;
		I50_SPARE_I306_7                        : BOOL;
		I60_ATC_DECLAMP_FB_I307_0               : BOOL;
		I60_ATC_CLAMP_FB_I307_1                 : BOOL;
		I60_ATC_STN_POKE_YOKE_1_I307_2          : BOOL;
		I60_ATC_STN_POKE_YOKE_2_I307_3          : BOOL;
		I60_ATC_STN_POKE_YOKE_3_I307_4          : BOOL;
		I60_ATC_STN_POKE_YOKE_4_I307_5          : BOOL;
		I60_ATC_SLAVE_MODL1_I307_6              : BOOL;
		I60_ATC_SLAVE_MODL2_I307_7              : BOOL;
		
		I70_DRUM_FEED_ALRM_I308_0              : BOOL;
		I70_SPARE_I308_1                        : BOOL;
		I70_DRUM_OFF_ON_I308_2                  : BOOL;
		I70_DRUM_CONV_REV_I308_3                : BOOL;
		I70_DRUM_CONV_FWD_I308_4                : BOOL;
		I70_SPARE_I308_5                        : BOOL;
		I70_SPARE_I308_6                        : BOOL;
		I70_SPARE_I308_7                        : BOOL;
		I80_ATC_DECLAMP_FB_I309_0               : BOOL;
		I80_ATC_CLAMP_FB_I309_1                 : BOOL;
		I80_ATC_STN_POKE_YOKE_1_I309_2          : BOOL;
		I80_ATC_STN_POKE_YOKE_2_I309_3          : BOOL;
		I80_ATC_STN_POKE_YOKE_3_I309_4          : BOOL;
		I80_ATC_STN_POKE_YOKE_4_I309_5          : BOOL;
		I80_ATC_SLAVE_MODL1_I309_6              : BOOL;
		I80_ATC_SLAVE_MODL2_I309_7              : BOOL;
		
		I80_SPARE_I310_0                        : BOOL;
		I80_SPARE_I310_1                        : BOOL;
		I80_SPARE_I310_2                        : BOOL;
		I80_SPARE_I310_3                        : BOOL;
		I80_SPARE_I310_4                        : BOOL;
		I80_SPARE_I310_5                        : BOOL;
		I80_SPARE_I310_6                        : BOOL;
		I80_SPARE_I310_7                        : BOOL;
		I80_SPARE_I311_0                        : BOOL;
		I80_SPARE_I311_1                        : BOOL;
		I80_SPARE_I311_2                        : BOOL;
		I80_SPARE_I311_3                        : BOOL;
		I80_SPARE_I311_4                        : BOOL;
		I80_SPARE_I311_5                        : BOOL;
		I80_SPARE_I311_6                        : BOOL;
		I80_SPARE_I311_7                        : BOOL;		
		
		O10_XTS_GREASE_VALVE_ON_Q300_0					: BOOL;
		O10A_SPARE_Q300_1								: BOOL;
		O10A_SPARE_Q300_2                               : Bool;
		O10A_SPARE_Q300_3                               : Bool;
		O10A_SPARE_Q300_4                               : Bool;
		O10A_SPARE_Q300_5                               : Bool;
		O10_BARLIGHT_OP1_Q300_6                         : Bool;
		O10_BARLIGHT_OP2_Q300_7                         : Bool;
		O10A_BDY_EMPT_CAM_LGHT1_ON_Q301_0               : Bool;
		O10A_BDY_EMPT_CAM_LGHT2_ON_Q301_1               : Bool;
		O10A_FIRTREE_ORING_CAM_LGHT1_ON_Q301_2          : Bool;
		O10A_FIRTREE_ORING_CAM_LGHT2_ON_Q301_3          : Bool;
		O10A_ORING_CAM_LGHT1_ON_Q301_4                  : Bool;
		O10A_ORING_CAM_LGHT2_ON_Q301_5                  : Bool;
		O10A_FIRTREE_ORING_CAMBAR_LGHT1_ON_Q301_6       : Bool;
		O10A_SPARE_Q301_7                               : Bool;
		
		O10B_DRUM_MTR_FWD_Q302_0                        : Bool;
		O10B_DRUM_RST_Q302_1                            : Bool;
		O10B_DRUM_EXT_SPEED_Q302_2                      : Bool;
		O10A_SPARE_Q302_3_Q302_3                        : Bool;
		O10B_DRUM_RUN_IND_Q302_4                        : Bool;
		O10_TWR_LMP_RD_Q302_5                           : Bool;
		O10_TWR_LMP_GN_Q302_6                           : Bool;
		O10_TWR_LMP_YELW_Q302_7                         : Bool;
		O10_TWR_LMP_BUZZ_Q303_0                         : Bool;
		O10B_SPARE_Q303_1 		                        : Bool;
		O10B_FIRTREE_ORING_CAM_LGHT1_ON_Q303_2          : Bool;
		O10B_FIRTREE_ORING_CAM_LGHT2_ON_Q303_3          : Bool;
		O10B_ORING_CAM_LGHT1_ON_Q303_4                  : Bool;
		O10B_ORING_CAM_LGHT2_ON_Q303_5                  : Bool;
		O10B_FIRTREE_ORING_CAMBAR_LGHT1_ON_Q303_6       : Bool;
		O10B_SPARE_Q303_7                               : BOOL;
		
		O20_SPARE_Q304_0                                : Bool;
		O20_SPARE_Q304_1                                : Bool;
		O20_SPARE_Q304_2                                : Bool;
		O20_SPARE_Q304_3                                : Bool;
		O30_DRUM_MTR_FWD_Q304_4                         : Bool;
		O30_DRUM_RST_Q304_5                             : Bool;
		O30_DRUM_EXT_SPEED_Q304_6                       : Bool;
		O30_SPARE_Q304_7_Q304_7                         : Bool;
		O30_DRUM_RUN_IND_Q305_0                         : Bool;
		O30_CAM_LGHT1_ON_Q305_1                         : Bool;
		O30_CAM_LGHT2_ON_Q305_2                         : Bool;
		O30_SPARE_Q305_3                                : Bool;
		O30_SPARE_Q305_4                                : Bool;
		O50_DRUM_MTR_FWD_Q305_5                         : Bool;
		O50_DRUM_RST_Q305_6                             : Bool;
		O50_SPARE_Q305_7                                : Bool;
		
		O50_DRUM_EXT_SPEED_Q306_0                       : Bool;
		O50_SPARE_Q306_1                                : Bool;
		O50_DRUM_RUN_IND_Q306_2                         : Bool;
		O50_CAM_LGHT1_ON_Q306_3                         : Bool;
		O50_CAM_LGHT2_ON_Q306_4                         : Bool;
		O50_SPARE_Q306_5                                : Bool;
		O50_SPARE_Q306_6                                : Bool;
		O50_BARLIGHT_OP1_Q306_7                         : Bool;
		O50_BARLIGHT_OP2_Q307_0                         : Bool;
		O70_DRUM_MTR_FWD_Q307_1                         : BOOL;
		O70_DRUM_RST_Q307_2                             : Bool;
		O70_DRUM_EXT_SPEED_Q307_3                       : Bool;
		O70_SPARE_Q307_4                                : Bool;
		O70_DRUM_RUN_IND_Q307_5                         : Bool;
		O70_CAM_LGHT1_ON_Q307_6                         : Bool;
		O70_CAM_LGHT2_ON_Q307_7                         : Bool;
		
		O70_BARLIGHT_OP1_Q308_0                         : Bool;
		O70_BARLIGHT_OP2_Q308_1                         : Bool;
		O70_SPARE_Q308_2                                : Bool;
		O70_SPARE_Q308_3                                : Bool;
		O70_SPARE_Q308_4                                : Bool;
		O70_SPARE_Q308_5                                : Bool;
		O70_SPARE_Q308_6                                : Bool;
		O70_SPARE_Q308_7                                : Bool;
		O70_SPARE_Q309_0                                : Bool;
		O70_SPARE_Q309_1                                : Bool;
		O70_SPARE_Q309_2                                : Bool;
		O70_SPARE_Q309_3                                : Bool;
		O70_SPARE_Q309_4                                : Bool;
		O70_SPARE_Q309_5                                : Bool;
		O70_SPARE_Q309_6                                : Bool;
		O70_SPARE_Q309_7                                : Bool;		
END_VAR

// ---- POUs/OP10_Profinet_IO/Master1_IO.TcGVL

VAR_GLOBAL
	
//port1
I10A_MAIN_AIR_PRES_FB_I1000_0					: BOOL;
I10A_SPARE_I1000_1                              : BOOL;
I10A_BDY_REJ_BIN_OVERFLW_I1000_2                : BOOL;
I10A_SPARE_I1000_3                              : BOOL;
I10A_SPARE_I1000_4                              : BOOL;
I10_LH_LNR_TRK_BDY_PRSN_I1000_5                 : BOOL;
I10_RH_LNR_TRK_BDY_PRSN_I1000_6                 : BOOL;
I10_LH_LNR_TRCK_FIX_CHO_1_I1000_7               : BOOL;

I10_LH_LNR_TRCK_FIX_CHO_2_I1001_0               : BOOL;
I10_RH_LNR_TRCK_FIX_CHO_1_I1001_1               : BOOL;
I10_RH_LNR_TRCK_FIX_CHO_2_I1001_2               : BOOL;
I10A_BDY1_PRSN_MOVER_I1001_3                    : BOOL;
I10A_BDY2_PRSN_MOVER_I1001_4                    : BOOL;
I10B_BDY1_PRSN_MOVER_I1001_5                    : BOOL;
I10B_BDY2_PRSN_MOVER_I1001_6                    : BOOL;
I10A_SPARE_I1001_7                              : BOOL;

//port2
I10A_DRUM_LH_CONV_OVR_FLW_I1010_0               : BOOL;
I10A_DRUM_RH_CONV_OVR_FLW_I1010_1               : BOOL;
I10A_ORING_LH_GRPR_CLSE_I1010_2                 : BOOL;
I10A_ORING_LH_GRPR_OPN_I1010_3                  : BOOL;
I10A_ORING_LH_PUSHR_CYL_REV_I1010_4             : BOOL;
I10A_ORING_RH_GRPR_OPN_I1010_5               	: BOOL;
I10A_ORING_RH_GRPR_CLSE_I1010_6             	: BOOL;
I10A_ORING_RH_PUSHR_CYL_REV_I1010_7       	    : BOOL;

I10A_ORING_ROTRY_CYL_O_DEG_I1011_0              : BOOL;
I10A_ORING_ROTRY_CYL_180_DEG_I1011_1            : BOOL;
I10A_ORING_HORZ_CYL_REV_I1011_2                 : BOOL;
I10A_ORING_HORZ_CYL_FWD_I1011_3                 : BOOL;
I10A_ORING_VERT_CYL_UP_I1011_4                  : BOOL;
I10A_ORING_VERT_CYL_DWN_I1011_5                 : BOOL;
I10A_LH_FIRTRE_ORING_REJ_CYL_REV_I1011_6        : BOOL;
I10A_LH_FIRTRE_ORING_REJ_CYL_FWD_I1011_7        : BOOL;

//port3
I10A_RH_FIRTRE_ORING_REJ_CYL_REV_I1020_0        : BOOL;
I10A_RH_FIRTRE_ORING_REJ_CYL_FWD_I1020_1        : BOOL;
I10A_BDY_SING_CYL_CLSE_I1020_2                  : BOOL;
I10A_BDY_SING_CYL_OPN_I1020_3                   : BOOL;
I10A_ORING_RH_GRPR_OPN_I1020_4                  : BOOL;
I10A_ORING_RH_PUSHR_CYL_FWD_I1020_5             : BOOL;
I10A_ORING_REJ_BIN_PRSNCE_I1020_6               : BOOL;
I10A_BOWL_TRK_INDXR_POS1_I1020_7                : BOOL;

I10A_BOWL_TRK_INDXR_POS2_I1021_0                : BOOL;
I10A_BOWL_TRK_INDXR_POS3_I1021_1                : BOOL;
I10A_SPARE_I1021_2                              : BOOL;
I10A_SPARE_I1021_3                              : BOOL;
I10A_SPARE_I1021_4                              : BOOL;
I10A_SPARE_I1021_5                              : BOOL;
I10A_SPARE_I1021_6                              : BOOL;
I10A_SPARE_I1021_7                              : BOOL;

//port4
I10B_DRUM_LH_CONV_OVR_FLW_I1030_0               : BOOL;
I10B_DRUM_RH_CONV_OVR_FLW_I1030_1               : BOOL;
I10B_ORING_LH_GRPR_CLSE_I1030_2                 : BOOL;
I10B_ORING_LH_GRPR_OPN_I1030_3                  : BOOL;
I10B_ORING_LH_PUSHR_CYL_REV_I1030_4             : BOOL;
I10B_ORING_RH_GRPR_OPN_I1030_5     		        : BOOL;
I10B_ORING_RH_GRPR_CLSE_I1030_6                 : BOOL;
I10B_ORING_RH_PUSHR_CYL_REV_I1030_7             : BOOL;

I10B_ORING_ROTRY_CYL_O_DEG_I1031_0              : BOOL;
I10B_ORING_ROTRY_CYL_180_DEG_I1031_1            : BOOL;
I10B_ORING_HORZ_CYL_REV_I1031_2                 : BOOL;
I10B_ORING_HORZ_CYL_FWD_I1031_3                 : BOOL;
I10B_ORING_VERT_CYL_UP_I1031_4                  : BOOL;
I10B_ORING_VERT_CYL_DWN_I1031_5                 : BOOL;
I10B_LH_FIRTRE_ORING_REJ_CYL_REV_I1031_6        : BOOL;
I10B_LH_FIRTRE_ORING_REJ_CYL_FWD_I1031_7        : BOOL;

//port5
I10B_RH_FIRTRE_ORING_REJ_CYL_REV_I1040_0        : BOOL;
I10B_RH_FIRTRE_ORING_REJ_CYL_FWD_I1040_1        : BOOL;
I10B_BDY_SING_CYL_CLSE_I1040_2                  : BOOL;
I10B_BDY_SING_CYL_OPN_I1040_3                   : BOOL;
I10B_ORING_RH_GRPR_OPN_I1040_4                  : BOOL;
I10B_ORING_RH_PUSHR_CYL_FWD_I1040_5             : BOOL;
I10B_ORING_REJ_BIN_PRSNCE_I1040_6               : BOOL;
I10B_BOWL_TRK_INDXR_POS1_I1040_7                : BOOL;

I10B_BOWL_TRK_INDXR_POS2_I1041_0                : BOOL;
I10B_BOWL_TRK_INDXR_POS3_I1041_1                : BOOL;
I10B_SPARE_I1041_2                              : BOOL;
I10B_SPARE_I1041_3                              : BOOL;
I10B_SPARE_I1041_4                              : BOOL;
I10B_SPARE_I1041_5                              : BOOL;
I10B_SPARE_I1041_6                              : BOOL;
I10B_SPARE_I1041_7                              : BOOL;

//port6
O10A_ORING_LH_GRPR_CLSE_OPN_Q1050_0             : BOOL;
O10A_ORING_LH_PUSHR_CYL_REV_FWD_Q1050_1         : Bool;
O10A_ORING_RH_GRPR_CLSE_OPN_Q1050_2             : Bool;
O10A_ORING_RH_PUSHR_CYL_REV_FWD_Q1050_3         : Bool;
O10A_ORING_ROTRY_CYL_O_DEG_Q1050_4              : Bool;
O10A_ORING_ROTRY_CYL_180_DEG_Q1050_5            : Bool;
O10A_ORING_HORZ_CYL_REV_Q1050_6                 : Bool;
O10A_ORING_HORZ_CYL_FWD_Q1050_7                 : BOOL;

O10A_ORING_VERT_CYL_UP_Q1051_0                  : BOOL;
O10A_ORING_VERT_CYL_DWN_Q1051_1                 : BOOL;
O10A_LH_FIRTRE_ORING_REJ_CYL_REV_Q1051_2        : Bool;
O10A_LH_FIRTRE_ORING_REJ_CYL_FWD_Q1051_3        : Bool;
O10A_RH_FIRTRE_ORING_REJ_CYL_REV_Q1051_4        : Bool;
O10A_RH_FIRTRE_ORING_REJ_CYL_FWD_Q1051_5        : Bool;
O10A_BDY_SING_CYL_CLSE_Q1051_6                  : Bool;
O10A_BDY_SING_CYL_OPN_Q1051_7                   : BOOL;

O10A_SPARE_Q1052_0                              : BOOL;
O10A_DRUM_FEED_AIRPURGE_ON_Q1052_1              : BOOL;
O10A_SPARE_Q1052_2                              : Bool;
O10A_SPARE_Q1052_3                              : Bool;
O10A_SPARE_Q1052_4                              : Bool;
O10A_SPARE_Q1052_5                              : Bool;
O10A_SPARE_Q1052_6                              : Bool;
O10A_SPARE_Q1052_7                              : BOOL;

O10A_SPARE_Q1053_0                              : BOOL;
O10A_SPARE_Q1053_1                              : Bool;
O10A_SPARE_Q1053_2                              : Bool;
O10A_SPARE_Q1053_3                              : Bool;
O10A_SPARE_Q1053_4                              : Bool;
O10A_SPARE_Q1053_5                              : Bool;
O10A_SPARE_Q1053_6                              : Bool;
O10A_SPARE_Q1053_7                              : BOOL;

//port7
O10B_ORING_LH_GRPR_CLSE_OPN_Q1060_0             : BOOL;
O10B_ORING_LH_PUSHR_CYL_REV_FWD_Q1060_1         : Bool;
O10B_ORING_RH_GRPR_CLSE_OPN_Q1060_2             : Bool;
O10B_ORING_RH_PUSHR_CYL_REV_FWD_Q1060_3         : Bool;
O10B_ORING_ROTRY_CYL_O_DEG_Q1060_4              : Bool;
O10B_ORING_ROTRY_CYL_180_DEG_Q1060_5            : Bool;
O10B_ORING_HORZ_CYL_REV_Q1060_6                 : Bool;
O10B_ORING_HORZ_CYL_FWD_Q1060_7                 : BOOL;

O10B_ORING_VERT_CYL_UP_Q1061_0                  : BOOL;
O10B_ORING_VERT_CYL_DWN_Q1061_1                 : Bool;
O10B_LH_FIRTRE_ORING_REJ_CYL_REV_Q1061_2        : Bool;
O10B_LH_FIRTRE_ORING_REJ_CYL_FWD_Q1061_3        : Bool;
O10B_RH_FIRTRE_ORING_REJ_CYL_REV_Q1061_4        : Bool;
O10B_RH_FIRTRE_ORING_REJ_CYL_FWD_Q1061_5        : Bool;
O10B_BDY_SING_CYL_CLSE_Q1061_6                  : Bool;
O10B_BDY_SING_CYL_OPN_Q1061_7                   : BOOL;

O10B_DRUM_FEED_AIRPURGE_ON_Q1062_0              : BOOL;
O10B_SPARE_Q1062_1                              : Bool;
O10B_SPARE_Q1062_2                              : Bool;
O10B_SPARE_Q1062_3                              : Bool;
O10B_SPARE_Q1062_4                              : Bool;
O10B_SPARE_Q1062_5                              : Bool;
O10B_SPARE_Q1062_6                              : Bool;
O10B_SPARE_Q1062_7                              : BOOL;

O10B_SPARE_Q1063_0                              : BOOL;
O10B_SPARE_Q1063_1                              : Bool;
O10B_SPARE_Q1063_2                              : Bool;
O10B_SPARE_Q1063_3                              : Bool;
O10B_SPARE_Q1063_4                              : Bool;
O10B_SPARE_Q1063_5                              : Bool;
O10B_SPARE_Q1063_6                              : Bool;
O10B_SPARE_Q1063_7                              : BOOL;

//port8
O20_LH_OIL_DISPN_ON_Q1150_0                     : BOOL;
O20_LH_OIL_SPIN_ON_Q1150_1                     : BOOL;
O20_RH_OIL_DISPN_ON_Q1150_2                      : BOOL;
O20_RH_OIL_SPIN_ON_Q1150_3                      : Bool;
O30_LH_REJ_CYL_REV_Q1150_4                      : BOOL;
O30_LH_REJ_CYL_FWD_Q1150_5                      : BOOL;
O30_RH_REJ_CYL_REV_Q1150_6                      : BOOL;
O30_RH_REJ_CYL_FWD_Q1150_7                      : BOOL;

O40_TOOL_CHO_UNLOCK_Q1151_0                     : Bool;
O40_TOOL_CHO_LOCK_Q1151_1                       : Bool;
O50_LH_GRIP_OPN_Q1151_2                         : BOOL;
O50_LH_GRIP_CLSE_Q1151_3                        : BOOL;
O50_RH_GRIP_OPN_Q1151_4                         : BOOL;
O50_RH_GRIP_CLSE_Q1151_5                        : BOOL;
O50_LH_REJ_CYL_REV_Q1151_6                      : BOOL;
O50_LH_REJ_CYL_FWD_Q1151_7                      : BOOL;

O50_RH_REJ_CYL_REV_Q1152_0                      : BOOL;
O50_RH_REJ_CYL_FWD_Q1152_1                      : BOOL;
O60_TOOL_CHO_UNLOCK_Q1152_2                     : Bool;
O60_TOOL_CHO_LOCK_Q1152_3                       : Bool;
O70_LH_REJ_CYL_REV_Q1152_4                      : BOOL;
O70_LH_REJ_CYL_FWD_Q1152_5                      : BOOL;
O70_RH_REJ_CYL_REV_Q1152_6                      : BOOL;
O70_RH_REJ_CYL_FWD_Q1152_7                      : BOOL;

O80_TOOL_CHO_UNLOCK_Q1153_0                     : BOOL;
O80_TOOL_CHO_LOCK_Q1153_1                       : Bool;
O30_AIR_PURGE_ON_Q1153_2                        : BOOL;
O30_SPARE_Q1153_3      	    	                : BOOL;
O50_AIR_PURGE_ON_Q1153_4                        : Bool;
O30_SPARE_Q1153_5 			                    : BOOL;
O70_AIR_PURGE_ON_Q1153_6                        : BOOL;
O30_SPARE_Q1153_7                               : Bool;
END_VAR

// ---- POUs/OP10_Profinet_IO/MASTER2_IO.TcGVL

VAR_GLOBAL
	//port1
I30_DRUM_FEED_CONV1_OVERFLW_I1100_0				 : BOOL;
I30_DRUM_FEED_CONV2_OVERFLW_I1100_1              : BOOL;
I30_LH_REJ_CYL_FWD_I1100_2                       : BOOL;
I30_LH_REJ_CYL_REV_I1100_3                       : BOOL;
I30_RH_REJ_CYL_FWD_I1100_4                       : BOOL;
I30_RH_REJ_CYL_REV_I1100_5                       : BOOL;
I30_TOP_REJ_BIN_PRSNCE_I1100_6                   : BOOL;
I30_BOT_REJ_BIN_PRSNCE_I1100_7                   : BOOL;

I50_DRUM_FEED_CONV1_OVERFLW_I1101_0              : BOOL;
I50_DRUM_FEED_CONV2_OVERFLW_I1101_1              : BOOL;
I50_LH_REJ_CYL_FWD_I1101_2                       : BOOL;
I50_LH_REJ_CYL_REV_I1101_3                       : BOOL;
I50_RH_REJ_CYL_FWD_I1101_4                       : BOOL;
I50_RH_REJ_CYL_REV_I1101_5                       : BOOL;
I50_SPARE_I1101_6                                : BOOL;
I50_LH_GRIP_CLSE_I1101_7                         : BOOL;

//port2
I50_SPARE_I1110_0                                : BOOL;
I50_RH_GRIP_CLSE_I1110_1                         : BOOL;
I70_DRUM_FEED_CONV1_OVERFLW_I1110_2              : BOOL;
I70_DRUM_FEED_CONV2_OVERFLW_I1110_3              : BOOL;
I70_LH_REJ_CYL_FWD_I1110_4                       : BOOL;
I70_LH_REJ_CYL_REV_I1110_5                       : BOOL;
I70_RH_REJ_CYL_FWD_I1110_6                       : BOOL;
I70_RH_REJ_CYL_REV_I1110_7                       : BOOL;

I50_TOP_REJ_BIN_PRSNCE_I1111_0                   : BOOL;
I50_BOT_REJ_BIN_PRSNCE_I1111_1                   : BOOL;
I70_TOP_REJ_BIN_PRSNCE_I1111_2                   : BOOL;
I70_BOT_REJ_BIN_PRSNCE_I1111_3                   : BOOL;
I70_SPARE_I1111_4                                : BOOL;
I70_SPARE_I1111_5                                : BOOL;
I70_SPARE_I1111_6                                : BOOL;
I70_SPARE_I1111_7                                : BOOL;



END_VAR

// ---- POUs/Programs/Error_GVL.TcGVL

VAR_GLOBAL
	berror: ARRAY [0..2001] OF BOOL;
	bclear: ARRAY [0..2001] OF BOOL;
	reset: BOOL;
END_VAR

// ---- POUs/Programs/OP110/OP110_GVL.TcGVL

VAR_GLOBAL
//GENERAL
OP110_Auto:					BOOL;
OP110_Mode_Ack:				BOOL;
OP110_HomeRunning:			BOOL;
OP110_ErrorActive:			BOOL;
OP110_Home_PB:				BOOL;
OP110_Work_PB:				BOOL;
OP110_ManualSafetyBypass:	BOOL;
OP110_LightCurtainBypass:	BOOL;
OP110_OperationCompleted:	BOOL;
OP110_LampCheck:				BOOL;
OP110_MachineLamp:			BOOL;
OP110_ComponentOk:			BOOL;
OP110_ComponentNok:			BOOL;
OP110_RepeatBit:				BOOL;
OP110_HomingResetBit:		BOOL;
OP110_ControlledByRobo:		BOOL;
OP110_Any_Bypass:			BOOL;
OP110_ManualModeStatus:		INT;
OP110_ManualModeWord:		INT;
OP110_AutoRunning:			BOOL;
OP110_StepRunning:			BOOL;
OP110_StartEnable:   		BOOL;
OP110_HomeConditionOK:		BOOL;
OP110_Temp_hmeOK:			BOOL;
OP110_Machine_Stop: 			BOOL;
OP110_AutoSeq:				INT;
OP110_LH_AutoSeq: 			INT;
OP110_RH_AutoSeq: 			INT;
OP110_Homing_Seq:			INT;
OP110_Safety_OK:				BOOL;
OP110_Stop_Request : BOOl;

Automatic_Run:				BOOL;    //from master mode block
Manual_mode: 				BOOL;    //from master mode block

OP110_Prev_Stat_Operation_Completed: BOOL;
OP110_Prev_Comp_Status: INT;
OP110_Prev_LH_COMP_OK:BOOL;
OP110_Prev_LH_COMP_NOK:BOOL;
OP110_Prev_RH_COMP_OK:BOOL;
OP110_Prev_RH_COMP_NOK:BOOL;
OP110_LH_Operation_Completed:BOOL;
OP110_RH_Operation_Completed:BOOL;


//Servo controls
	OP110_Servo_Enable	: BOOL;
	OP110_Servo_Reset	: BOOL;
	SR110_Vert_servo_not_Home: BOOL;
	SR110_Vert_servo: FB_Axis;
	
//ModeSelection Outputs
//OP130_AutoSelected:		    BOOL;
OP110_ManualSelected:		BOOL;
OP110_StepSelected:			BOOL;
OP110_AutoSelected:		    BOOL;


//HMI Tags(From HMI)
OP110_HMI_AutoMode:						BOOL;
OP110_HMI_ManualMode:					BOOL;
OP110_HMI_StepMode:						BOOL;
OP110_HMI_CycleStart:					BOOL;


OP110_HMI_Homing:						BOOL;
SR20_Vert_Servo_Max_Lim:				BOOL;
OP110_HMI_Jog_Pos: BOOL;
OP110_HMI_Jog_Neg: BOOL;

OP110_AUTO_STP_NO: INT;

// MANUAL
		
// AUTO	
		// FROM MASTER CONTROL BLOCK
	OP110_FIXTURE_2					: INT;               //For the comp status in the fixture
	OP110_FIXTURE_1					: INT; 				 //For the comp status in the fixture
// SERVO VARIABLE
	OP110_VERT_SERVO_STRT			: BOOL;				// SERVO MOVE TO TARGET POSITION
	OP110_SERVO_POS_DONE				: BOOL;				// SERVO POSITION REACHED
	OP110_SERVO_ON_SFE_WRK			: BOOL;				// SERVO ACTUAL POSITION = SERVO SAFE POSITION
	OP110_SERVO_ON_WRK				: BOOL;				// SERVO ACTUAL POSITION = SERVO WORK POSITION
	OP110_SERVO_ON_HOME				: BOOL;				// SERVO ACTUAL POSITION = SERVO HOME POSITION	
	
	OP110_VERT_SERVO_HME_POS			: REAL := 0;         // SERVO IN HOME POSITION
	OP110_VERT_SERVO_POSITION		: LREAL ;			// SERVO ACTUAL POSITION
	OP110_VERT_SERVO_SFE_WRK_POS		: REAL := 40;		// SERVO SAFE WORK POSITION FROM RECEIPE
	OP110_VERT_SERVO_WRK_POS			: REAL := 200;		// SERVO WORK POSITION FROM RECEIPE	
	OP110_VERT_SERVO_TARGET			: REAL;				// SERVO AUTO TARGET POSITION

END_VAR

VAR_GLOBAL PERSISTENT
	
// MANUAL
	OP110_STN_ENABLE				: BOOL;		
	OP110_OIL_TIMER 				: INT;
	OP110_STN_RUNNING 				: BOOL;
// AUTO
	OP110_BYPASS					: BOOL;				// OP110 ON-BYPASS / OFF-NOT BYPASSED
	OP110_LH_OIL_OK					: BOOL;				// TO MASTER CONTROL BLOCK OILLING LH OK BIT
	OP110_LH_OIL_NOK				: BOOL;				// TO MASTER CONTROL BLOCK OILLING LH NOK BIT
	OP110_RH_OIL_OK					: BOOL;				// TO MASTER CONTROL BLOCK OILLING RH OK BIT
	OP110_RH_OIL_NOK				: BOOL;				// TO MASTER CONTROL BLOCK OILLING RH NOK BIT
	
//Setting Parameters
    OP110_HMI_Servo_Speed    	: REAL;
    OP110_HMI_Low_Limit		 	: REAL;
    OP110_HMI_High_Limit	 	: REAL;
	OP110_HMI_Safe_Home		 	: REAL;
	OP110_HMI_Safe_Work		 	: REAL;
	OP110_Oil_Position_Offset	: REAL :=10;
	OP110_Oiling_Velocity		: REAL :=20;
//Error
OP110_ErrorWord_0: DINT;
OP110_ErrorWord_1: DINT;
OP110_ErrorWord_2: DINT;

	OP110_Cycle_time: UDINT;	
	
END_VAR

// ---- POUs/Programs/OP110/OP110_HMI_GVL.TcGVL

VAR_GLOBAL
	
SR110_Vert_servo_ctrl:Servo_Control;
	SR110_Vert_servo_status:stManualModeAxis;
	OP110_HMI_Reset:						    BOOL;
END_VAR

// ---- POUs/Programs/OP110/OP110_Recipe.TcGVL

VAR_GLOBAL PERSISTENT
	OP110_DLY_OIL_ON : INT;
	OP110_VERT_SERVO_WORK_POS : REAL;
	OP110_VERT_SERVO_SFE_WORK_POS : REAL;	
END_VAR

// ---- POUs/Programs/OP130/OP130_GVL.TcGVL

VAR_GLOBAL
	//GENERAL
OP130_Auto:					BOOL;
OP130_HomeRunning:			BOOL;
OP130_ErrorActive:			BOOL;
OP130_Home_PB:				BOOL;
OP130_Work_PB:				BOOL;
OP130_ManualSafetyBypass:	BOOL;
OP130_LightCurtainBypass:	BOOL;
OP130_OperationCompleted:	BOOL;
OP130_LampCheck:			BOOL;
OP130_MachineLamp:			BOOL;
OP130_ComponentOk:			BOOL;
OP130_ComponentNok:			BOOL;
OP130_RepeatBit:			BOOL;
OP130_HomingResetBit:		BOOL;
OP130_ControlledByRobo:		BOOL;
OP130_Any_Bypass:			BOOL;
OP130_ManualModeStatus:		INT;
OP130_ManualModeWord:		INT;
OP130_AutoRunning:			BOOL;
OP130_StepRunning:			BOOL;
OP130_StartEnable:   		BOOL;
OP130_Machine_Stop: 		BOOL;
OP130_AutoSeq:				INT;
OP130_LH_AutoSeq: 			INT;
OP130_RH_AutoSeq: 			INT;
OP130_Homing_Seq:			INT;
OP130_RH_Homing_Seq:		INT;
OP130_STN_MOVER				: INT;
OP130_Dry_Run:				BOOL;
OP130_LH_HomeOK:			BOOL;
OP130_RH_HomeOK:			BOOL;
//Automatic_Run:				BOOL;
OP130_Prev_Stat_Operation_Completed: BOOL;
OP130_Prev_Comp_Status: INT;
OP130_Prev_LH_COMP_OK:BOOL;
OP130_Prev_LH_COMP_NOK:BOOL;
OP130_Prev_RH_COMP_OK:BOOL;
OP130_Prev_RH_COMP_NOK:BOOL;
OP130_LH_Operation_Completed:BOOL;
OP130_RH_Operation_Completed:BOOL;

OP130_LH_Comp_OK: BOOL;
OP130_LH_Comp_NOK: BOOL;
OP130_RH_Comp_OK: BOOL;
OP130_RH_Comp_NOK: BOOL;
//ModeSelection Outputs
//OP130_AutoSelected:		    BOOL;
OP130_ManualSelected:		BOOL;
OP130_StepSelected:			BOOL;
OP130_AutoSelected:		    BOOL;
OP130_Temp_Home_OK:			BOOL;
OP130_Home_ConditionOK:		BOOL;
OP130_OperationEnable:		BOOL;
OP130_SafetyNoerror:		BOOL;

//Manual Cylinder FB Tags
CR130_RH_Rotart_Cyl_Status:	 INT;
CR130_LH_Rotart_Cyl_Status:	 INT;


//Manual Control Inputs

	CR130_LH_Rot_Cyl: Cylinder_Block_FOR_OP130;
	CR130_RH_Rot_Cyl: Cylinder_Block_FOR_OP130;
	SR130_LH_Vert_Servo: FB_Axis;
	SR130_RH_Vert_Servo: FB_Axis;
	
	SR130_Clm_Stepper: FB_Axis_FESTO;
	SR130_LH_Vert_Servo_Axis:AXIS_REF;
	SR130_RH_Vert_Servo_Axis:AXIS_REF;
	SR130_Clm_Stepper_Axis:AXIS_REF;
	SR130_LH_Servo_Control:Servo_Control;
	SR130_RH_Servo_Control:Servo_Control;
	SR130_Stepper_Control:Servo_Control;

	SR130_stManualModeAxis_LH_Vert_Servo:stManualModeAxis;
	SR130_stManualModeAxis_RH_Vert_Servo:stManualModeAxis;
	SR130_stManualModeAxis_Clamp_Stepper:stManualModeAxis;
	SR130_LH_Abs_Move_Start:BOOL;
	SR130_RH_Abs_Move_Start:BOOL;
//HMI Tags(From HMI)
OP130_HMI_AutoMode:						BOOL;
OP130_HMI_ManualMOde:					BOOL;
OP130_HMI_StepMode:						BOOL;
OP130_HMI_CycleStart:					BOOL;
OP130_HMI_LH_Rotary_Cyl_Home_PB:			BOOL;
OP130_HMI_LH_Rotary_Cyl_Work_PB:			BOOL;
OP130_HMI_RH_Rotary_Cyl_Home_PB:			BOOL;
OP130_HMI_RH_Rotary_Cyl_Work_PB:			BOOL;
OP130_HMI_Cycle_Start:					BOOL;
OP130_HMI_Reset:						BOOL;
OP130_HMI_Homing:						BOOL;

SR130_RH_Vert_Servo_Max_Lim:					LREAL;

SR130_RH_Vert_Servo_Min_Lim:					LREAL;
SR130_Clm_Vert_Max_Lim:					LREAL;


 

 		// Servo Positions
SR130_LH_Servo_Home_Position: 				LREAL;
SR130_LH_Servo_Home_Velocity: 				LREAL;
//SR130_HMI_LH_Servo_Work_Position:			LREAL;
//SR130_HMI_LH_Servo_Work_Velocity:			LREAL;
//SR130_HMI_LH_Servo_Lock_Position:			LREAL;
//SR130_HMI_LH_Servo_Lock_Velocity:			LREAL;
//SR130_HMI_LH_Servo_Rotation_Position:		LREAL;
//SR130_HMI_LH_Servo_Rotation_Velocity:		LREAL;
//SR130_HMI_LH_Servo_Torque_Low_Limit:			LREAL;
//SR130_HMI_LH_Servo_Torque_High_Limit:			LREAL;
//
SR130_RH_Servo_Home_Position: 				LREAL;
SR130_RH_Servo_Home_Velocity: 				LREAL;
//SR130_HMI_RH_Servo_Work_Position:			LREAL;
//SR130_HMI_RH_Servo_Work_Velocity:			LREAL;
//SR130_HMI_RH_Servo_Lock_Position:			LREAL;
//SR130_HMI_RH_Servo_Lock_Velocity:			LREAL;
//SR130_HMI_RH_Servo_Rotation_Position:		LREAL;
//SR130_HMI_RH_Servo_Rotation_Velocity:		LREAL;
//SR130_HMI_RH_Servo_Torque_Low_Limit:			LREAL;
//SR130_HMI_RH_Servo_Torque_High_Limit:			LREAL;


SR130_Stepper_Home_Position:				LREAL;
SR130_Stepper_Home_Velocity:				LREAL;
SR130_Stepper_Work_Position: 				LREAL;
SR130_Stepper_Work_Velocity: 				LREAL;






//Error
OP130_ErrorWord_0:    							 DINT;
OP130_ErrorWord_1:								 DINT;
OP130_ErrorWord_2:								 DINT;


//Recipe Tags

	
		//RH Servo
SR130_HMI_RH_Servo_Work_Position:			LREAL;
SR130_HMI_RH_Servo_Work_Velocity:			LREAL;
SR130_HMI_RH_Servo_Lock_Position:			LREAL;
SR130_HMI_RH_Servo_Lock_Velocity:			LREAL;
SR130_HMI_RH_Servo_Rotation_Position:		LREAL;
SR130_HMI_RH_Servo_Rotation_Velocity:		LREAL;
SR130_HMI_RH_Servo_Torque_Low_Limit:		LREAL;
SR130_HMI_RH_Servo_Torque_High_Limit:		LREAL;
SR130_HMI_RH_Servo_CylWork_Position:		LREAL;
SR130_HMI_RH_Servo_CylWork_Velocity:		LREAL;
SR130_HMI_RH_Servo_CylHome_Position:		LREAL;
SR130_HMI_RH_Servo_CylHome_Velocity:		LREAL;

OP130_Torque_Monitor_Time:TIME;




	OP130_Cycle_Time_Start: BOOL;
	OP130_Cycle_Time_Stop: BOOL;
	
	SR130_LH_Servo_Halt_Cmd:BOOL;
	SR130_RH_Servo_Halt_Cmd:BOOL;
OP130_STN_ENABLE: BOOL;
	
END_VAR
VAR_GLOBAL PERSISTENT
	// Servo
SR130_HMI_Servo_Work_Position:			LREAL;
SR130_HMI_Servo_Work_Velocity:			LREAL;
SR130_HMI_Servo_Lock_Position:			LREAL;
SR130_HMI_Servo_Lock_Velocity:			LREAL;
SR130_HMI_Servo_Rotation_Position:		LREAL;
SR130_HMI_Servo_Rotation_Velocity:		LREAL;
SR130_HMI_Servo_Torque_Low_Limit:		LREAL;
SR130_HMI_Servo_Torque_High_Limit:		LREAL;
SR130_HMI_Servo_CylWork_Position:		LREAL;
SR130_HMI_Servo_CylWork_Velocity:		LREAL;
SR130_HMI_Servo_CylHome_Position:		LREAL;
SR130_HMI_Servo_CylHome_Velocity:		LREAL;
SR130_LH_Vert_Servo_Max_Limit:			LREAL;
SR130_LH_Vert_Servo_Min_Lim:			LREAL;
SR130_Servo_Home_Position:				LREAL;
SR130_Servo_Home_Velocity:				LREAL;

//Torque limit

OP130_HMI_Pull_LOw_Torque_Limit: INT;
	OP130_HMI_Pull_High_Torque_Limit: INT;
	OP130_HMI_Pull_Torque_Limit:LREAL;
	
END_VAR

// ---- POUs/Programs/OP140/OP140_GVL.TcGVL

VAR_GLOBAL
	//GENERAL
OP140_DryRun				:BOOL;
OP140_Auto:					BOOL;
OP140_HomeRunning:			BOOL;
OP140_ErrorActive:			BOOL;
OP140_Home_PB:				BOOL;
OP140_Work_PB:				BOOL;
OP140_ManualSafetyBypass:	BOOL;
OP140_LightCurtainBypass:	BOOL;
OP140_OperationCompleted:	BOOL;
OP140_LampCheck:			BOOL;
OP140_MachineLamp:			BOOL;
OP140_ComponentOk:			BOOL;
OP140_ComponentNok:			BOOL;
OP140_RepeatBit:			BOOL;
OP140_HomingResetBit:		BOOL;
OP140_ControlledByRobo:		BOOL;
OP140_Any_Bypass:			BOOL;
OP140_ManualModeStatus:		INT;
OP140_ManualModeWord:		INT;
OP140_AutoRunning:			BOOL;
OP140_StepRunning:			BOOL;
OP140_StartEnable  :        BOOL;
OP140_StartEnable_1:   		BOOL;
OP140_StartEnable_2:   		BOOL;
OP140_StartEnable_3:   		BOOL;
OP140_Machine_Stop : 		BOOL;
OP140_TOOL_CHANGE_MODE_SELECTED: BOOL;


OP140_Homing_Seq   :		INT;

//Automatic_Run:				BOOL;

//auto 1
OP140A1_Prev_LH_COMP_OK:BOOL;
OP140A1_Prev_LH_COMP_NOK:BOOL;
OP140A1_Prev_RH_COMP_OK:BOOL;
OP140A1_Prev_RH_COMP_NOK:BOOL;
OP140A1_LH_Comp_OK: BOOL;
OP140A1_LH_Comp_NOK: BOOL;
OP140A1_RH_Comp_OK: BOOL;
OP140A1_RH_Comp_NOK: BOOL;

//auto 2
OP140A2_Prev_LH_COMP_OK:BOOL;
OP140A2_Prev_LH_COMP_NOK:BOOL;
OP140A2_Prev_RH_COMP_OK:BOOL;
OP140A2_Prev_RH_COMP_NOK:BOOL;
OP140A2_LH_Comp_OK: BOOL;
OP140A2_LH_Comp_NOK: BOOL;
OP140A2_RH_Comp_OK: BOOL;
OP140A2_RH_Comp_NOK: BOOL;

//auto 3

OP140A3_Prev_LH_COMP_OK:BOOL;
OP140A3_Prev_LH_COMP_NOK:BOOL;
OP140A3_Prev_RH_COMP_OK:BOOL;
OP140A3_Prev_RH_COMP_NOK:BOOL;
OP140A3_LH_Comp_OK: BOOL;
OP140A3_LH_Comp_NOK: BOOL;
OP140A3_RH_Comp_OK: BOOL;
OP140A3_RH_Comp_NOK: BOOL;




//LH ATEQ Tags:
OP140_LH_ATEQ_Result_Completed:BOOL;
OP140_RH_ATEQ_Result_Completed:BOOL;

//ModeSelection Outputs
//OP140_AutoSelected:		    BOOL;
OP140_ManualSelected:		BOOL;
OP140_StepSelected:			BOOL;
OP140_AutoSelected:		    BOOL;
OP140_Temp_Home_Ok:			BOOL;
OP140_Safety_No_Error:		BOOL;
OP140_HomeConditionOK:		BOOL;

//Manual Cylinder FB Tags
CR140_Horz_Cyl_1_Status:	 INT;
CR140_Horz_Cyl_2_Status:	 INT;
CR140_Horz_Cyl_3_Status:	 INT;
CR140_Vert_Cyl_1_Status:	 INT;
CR140_Vert_Cyl_2_Status:	 INT;
CR140_Vert_Cyl_3_Status:	 INT;
CR140_Wipe_Cyl_1_Status:	 INT;
CR140_Wipe_Cyl_2_Status:	 INT;
CR140_Wipe_Cyl_3_Status:	 INT;

//CR130_LH_Rotart_Cyl_Status:	 INT;

CR140_Horz_Cyl_1: Cylinder_Block;
	CR140_Horz_Cyl_2: Cylinder_Block;
	CR140_Horz_Cyl_3: Cylinder_Block;
	CR140_Vert_Cyl_1: Cylinder_Block;
	CR140_Vert_Cyl_2: Cylinder_Block;
	CR140_Vert_Cyl_3: Cylinder_Block;
	CR140_Top_Wipe_Cyl_1: Cylinder_Block;
	CR140_Top_Wipe_Cyl_2: Cylinder_Block;
	CR140_Top_Wipe_Cyl_3: Cylinder_Block;
	SR140_Vert_Servo_1: FB_Axis;
	SR140_Vert_Servo_2: FB_Axis;
	SR140_Vert_Servo_3: FB_Axis;
	SR140_HMI_Vert_Servo_MC1:stManualModeAxis;
	SR140_HMI_Vert_Servo_MC2:stManualModeAxis;
	
	SR140_Vert_Servo_Axis_1: Axis_ref;
	SR140_Vert_Servo_AXis_2: Axis_ref;
	SR140_Vert_Servo_Axis_3:Axis_ref;
	
	SR140_Vert_Servo_Ctrl_1: Servo_Control;
	SR140_Vert_Servo_Ctrl_2:Servo_Control;
//ATEQ Manual HMI Tags
OP140_ATEQ_SEL_NO :INT;
OP140_ATEQ_Start  :BOOL;
OP140_ATEQ_Reset  :BOOL;
OP140_ATEQ_Prog_No:INT;
OP140_ATEQ_Result_Ok  :BOOL;
OP140_ATEQ_Result_NOk  :BOOL;
OP140_STN_ENABLE_1: BOOL;
OP140_STN_ENABLE_2: BOOL;
OP140_STN_ENABLE_3: BOOL;
//ATEQ INPUTS and OUTPUTS
	 OP140_ATEQ1_Auto_Start:BOOL;
	 OP140_ATEQ2_Auto_Start:BOOL;
	 OP140_ATEQ3_Auto_Start:BOOL;
	 OP140_ATEQ4_Auto_Start:BOOL;
	 OP140_ATEQ5_Auto_Start:BOOL;
	 OP140_ATEQ6_Auto_Start:BOOL;
	 OP140_ATEQ1_Auto_Prog_No:INT;
	 OP140_ATEQ2_Auto_Prog_No:INT;
	 OP140_ATEQ3_Auto_Prog_No:INT;
	 OP140_ATEQ4_Auto_Prog_No:INT;
	 OP140_ATEQ5_Auto_Prog_No:INT;
	 OP140_ATEQ6_Auto_Prog_No:INT;
//LEAK FB Prog NO OUt

//HMI Tags(From HMI)
OP140_HMI_AutoMode:						BOOL;
OP140_HMI_ManualMOde:					BOOL;
OP140_HMI_StepMode:						BOOL;
OP140_HMI_CycleStart:					BOOL;
OP140_HMI_Horz_Cyl1_Home_PB:			BOOL;
OP140_HMI_Horz_Cyl1_Work_PB:			BOOL;
OP140_HMI_Horz_Cyl2_Home_PB:			BOOL;
OP140_HMI_Horz_Cyl2_Work_PB:			BOOL;
OP140_HMI_Horz_Cyl3_Home_PB:			BOOL;
OP140_HMI_Horz_Cyl3_Work_PB:			BOOL;
OP140_HMI_Vert_Cyl1_Home_PB:			BOOL;
OP140_HMI_Vert_Cyl1_Work_PB:			BOOL;
OP140_HMI_Vert_Cyl2_Home_PB:			BOOL;
OP140_HMI_Vert_Cyl2_Work_PB:			BOOL;
OP140_HMI_Vert_Cyl3_Home_PB:			BOOL;
OP140_HMI_Vert_Cyl3_Work_PB:			BOOL;
OP140_HMI_Wipe_Cyl1_Home_PB:			BOOL;
OP140_HMI_Wipe_Cyl1_Work_PB:			BOOL;
OP140_HMI_Wipe_Cyl2_Home_PB:			BOOL;
OP140_HMI_Wipe_Cyl2_Work_PB:			BOOL;
OP140_HMI_Wipe_Cyl3_Home_PB:			BOOL;
OP140_HMI_Wipe_Cyl3_Work_PB:			BOOL;
OP140_HMI_Cycle_Start:					BOOL;
OP140_HMI_Homing:						BOOL;

SR130_Vert_Servo_Work_vel:BOOL;

//LeakTestFB Tags
OP140_Leak1_Seq_Start:BOOL;
OP140_Leak1_Seq_Completed:BOOL;
OP140_Leak2_Seq_Start:BOOL;
OP140_Leak2_Seq_Completed:BOOL;
OP140_Leak3_Seq_Start:BOOL;
OP140_Leak3_Seq_Completed:BOOL;

//Error
OP140_ErrorWord_0:    							 DINT;
OP140_ErrorWord_1:								 DINT;
OP140_ErrorWord_2:								 DINT;

OP140_HMI_Vert4_Work_Pos:LREAL;
OP140_HMI_Vert4_Work_Vel:LREAL;
OP140_HMI_Vert5_Work_Pos:LREAL;
OP140_HMI_Vert5_Work_Vel:LREAL;
OP140_HMI_Vert6_Work_Pos:LREAL;
OP140_HMI_Vert6_Work_Vel:LREAL;

	OP140_ATEQ1_ResultCompleted:BOOL;
	 OP140_ATEQ2_ResultCompleted:BOOL;
	 OP140_ATEQ3_ResultCompleted:BOOL;
	 OP140_ATEQ4_ResultCompleted:BOOL;
	 OP140_ATEQ5_ResultCompleted:BOOL;
	 OP140_ATEQ6_ResultCompleted:BOOL;
     OP140_ATEQ1_ResultOK:BOOL;
	 OP140_ATEQ2_ResultOK:BOOL;
	 OP140_ATEQ3_ResultOK:BOOL;
	 OP140_ATEQ4_ResultOK:BOOL;
	 OP140_ATEQ5_ResultOK:BOOL;
	 OP140_ATEQ6_ResultOK:BOOL;
	 OP140_ATEQ1_ResultNOK:BOOL;
	 OP140_ATEQ2_ResultNOK:BOOL;
	 OP140_ATEQ3_ResultNOK:BOOL;
	 OP140_ATEQ4_ResultNOK:BOOL;
	 OP140_ATEQ5_ResultNOK:BOOL;
	 OP140_ATEQ6_ResultNOK:BOOL;
	 
	
	OP140_Servo1_Safety:BOOL;
	OP140_Servo2_Safety:BOOL;
	OP140_Servo3_Safety:BOOL;
	
	
	//ATEQ
	OP140_ATEQ1_Auto_Prog_No_out: INT;
	OP140_ATEQ2_Auto_Prog_No_out: INT;
	OP140_ATEQ3_Auto_Prog_No_out: INT;
	OP140_ATEQ4_Auto_Prog_No_out: INT;
	OP140_ATEQ5_Auto_Prog_No_out: INT;
	OP140_ATEQ6_Auto_Prog_No_out: INT;
	
	OP140_STN_MOVER: int;
END_VAR

VAR_GLOBAL PERSISTENT
	anvar: BOOL;
	//Recipe Tags

OP140_HMI_Vert1_Work_Pos:LREAL;
OP140_HMI_Vert1_Work_Vel:LREAL;
OP140_HMI_Vert2_Work_Pos:LREAL;
OP140_HMI_Vert2_Work_Vel:LREAL;
OP140_HMI_Vert3_Work_Pos:LREAL;
OP140_HMI_Vert3_Work_Vel:LREAL;
OP140_ATEQ_Test_Prog1_No:INT;
OP140_ATEQ_Test_Prog2_No:INT;
SR140_Vert_Servo_Max_Lim:					LREAL;
SR140_Vert_Servo_Min_Lim:					LREAL;
OP140_HMI_Vert_SafeWork_Pos:LREAL;
OP140_HMI_Vert1_SafeWork_Vel:LREAL;
OP140_HMI_Vert_Home_Pos:LREAL;
OP140_HMI_Vert_Home_Vel:LREAL;
OP140_HMI_Vert_SafeHome_Pos:LREAL;
OP140_HMI_Vert_SafeHome_Vel:LREAL;
END_VAR

// ---- POUs/Programs/OP140/OP140_HMI_GVL.TcGVL
//{attribute 'qualified_only'}
VAR_GLOBAL
	

OP140_HMI_Reset							:BOOL;
SR140_Vert_Servo_Ctrl_3					:Servo_Control;
SR140_HMI_Vert_Servo_MC3				:stManualModeAxis;


	OP140_ATEQ1_Result : STRING;
	OP140_ATEQ2_Result : STRING;
	OP140_ATEQ3_Result : STRING;
	OP140_ATEQ4_Result : STRING;
	OP140_ATEQ5_Result : STRING;
	OP140_ATEQ6_Result : STRING;
	
    OP140_ATEQ1_Status : STRING;
    OP140_ATEQ2_Status : STRING;
    OP140_ATEQ3_Status : STRING;
    OP140_ATEQ4_Status : STRING;
    OP140_ATEQ5_Status : STRING;
    OP140_ATEQ6_Status : STRING;
	 
	OP140_ATEQ1_Prgrm_Num : STRING; 
	OP140_ATEQ2_Prgrm_Num : STRING; 
	OP140_ATEQ3_Prgrm_Num : STRING; 
	OP140_ATEQ4_Prgrm_Num : STRING; 
	OP140_ATEQ5_Prgrm_Num : STRING; 
	OP140_ATEQ6_Prgrm_Num : STRING; 
END_VAR

// ---- POUs/Programs/OP150/OP150_GVL.TcGVL

VAR_GLOBAL
	
OP150A_LH_Start : BOOL;
OP150A_RH_Start : BOOL;
OP150B_LH_Start : BOOL;
OP150B_RH_Start : BOOL;
OP150C_LH_Start : BOOL;
OP150C_RH_Start : BOOL;

OP150_Lsr_Ready				    : BOOL;
OP150_Laser_Start		        : BOOL;
OP150_Lsr_Job_Change_Start      : BOOL;
OP150_Lsr_Job_Change_Complete   : BOOL;
OP150_Lsr_Text_Change_Start     : BOOL;
OP150_Lsr_Text_Change_Complete  : BOOL;	
OP150_Laser_Completed   		: BOOL;
OP150_Laser_Failed      		: BOOL;	
OP150_Lsr_Job_ID  				: UDINT;
OP150_Lsr_Block_ID 				: UDINT;
OP150_Lsr_String				: STRING[80];


OP150_A_ErrorActive			: BOOL;
OP150_B_ErrorActive			: BOOL;
OP150_C_ErrorActive			: BOOL;

OP150_ManualSelected	:BOOL;
OP150_StepSelected      :BOOL;
OP150_AutoSelected		:BOOL;
OP150_AutoRunning 		:BOOL;
OP150_StepRunning		:BOOL;
OP150_StartEnable		:BOOL;
OP150_Machine_Stop		:BOOL;

OP150_MoverPresent		: BOOL;
OP150_Temp_Home_OK		: BOOL;
OP150_HomeCondition_OK	: BOOL;
OP150_OperationEnable	: BOOL;

//HMI Tags(From HMI)
OP150_HMI_AutoMode:						BOOL;
OP150_HMI_ManualMOde:					BOOL;
OP150_HMI_StepMode:						BOOL;
OP150_HMI_CycleStart_PB:				BOOL;
OP150_HMI_Homing_PB:					BOOL;
OP150_HMI_Reset	:	 					BOOL;
//Mover Bit




END_VAR

VAR_GLOBAL PERSISTENT
	OP150A_LH_CMP_OK :BOOL;
	OP150A_RH_CMP_OK :BOOL;
	
	Laser_Line1 : STRING :='E2525';	 
	Laser_Line2 : STRING :='D7.89';  
	Laser_Line3 : STRING :='>PK25D<';
	
	OP150_Model				: STRING :='7.89';
END_VAR

// ---- POUs/Programs/OP160/OP160_GVL.TcGVL

VAR_GLOBAL
	//GENERAL
OP160_Auto:					BOOL;
OP160_HomeRunning:			BOOL;
OP160_ErrorActive:			BOOL;
OP160_Home_PB:				BOOL;
OP160_Work_PB:				BOOL;
OP160_ManualSafetyBypass:	BOOL;
OP160_LightCurtainBypass:	BOOL;
OP160_OperationCompleted:	BOOL;
OP160_LampCheck:			BOOL;
OP160_MachineLamp:			BOOL;
OP160_ComponentOk:			BOOL;
OP160_ComponentNok:			BOOL;
OP160_RepeatBit:			BOOL;
OP160_HomingResetBit:		BOOL;
OP160_ControlledByRobo:		BOOL;
OP160_Any_Bypass:			BOOL;
OP160_STN_MOVER: INT;
OP160_STN_ENABLE: BOOL;
OP160_ManualModeStatus:		INT;
OP160_ManualModeWord:		INT;
OP160_AutoRunning:			BOOL;
OP160_StepRunning:			BOOL;
OP160_StartEnable:   		BOOL;
OP160_Machine_Stop: 		BOOL;
OP160_AutoSeq:				INT;
OP160_LH_AutoSeq: 			INT;
OP160_RH_AutoSeq: 			INT;
OP160_Homing_Seq:			INT;
OP160_DryRun:				BOOL;
//Automatic_Run:				BOOL;
OP160_Prev_Stat_Operation_Completed: BOOL;
OP160_Prev_Comp_Status: INT;
OP160_Prev_LH_COMP_OK:BOOL;
OP160_Prev_LH_COMP_NOK:BOOL;
OP160_Prev_RH_COMP_OK:BOOL;
OP160_Prev_RH_COMP_NOK:BOOL;
OP160_LH_Operation_Completed:BOOL;
OP160_RH_Operation_Completed:BOOL;

OP160_LH_Comp_OK: BOOL;
OP160_LH_Comp_NOK: BOOL;
OP160_RH_Comp_OK: BOOL;
OP160_RH_Comp_NOK: BOOL;

OP160_RH_Laser_Start:BOOL;
OP160_LH_Laser_Start:BOOL;
OP160_RH_Laser_Completed:BOOL;
OP160_LH_Laser_Completed:BOOL;

//ModeSelection Outputs
//OP160_AutoSelected:		    BOOL;

OP160_ManualSelected:		BOOL;
OP160_StepSelected:			BOOL;
OP160_AutoSelected:		    BOOL;
OP160_HomeCondition_OK:BOOL;
OP160_Temp_Home_OK:BOOL;

//Manual Cylinder FB Tags

CR130_RH_Rotart_Cyl_Status:	 INT;
CR130_LH_Rotart_Cyl_Status:	 INT;

// Manual Cyl

CR160_Gripper_Cyl_1: Cylinder_Block;
CR160_Gripper_Cyl_2:Cylinder_Block;

CR160_MoverREM_Cyl: Cylinder_Block;
//HMI Tags(From HMI)

OP160_HMI_AutoMode:						BOOL;
OP160_HMI_ManualMOde:					BOOL;
OP160_HMI_StepMode:						BOOL;
OP160_HMI_CycleStart:					BOOL;
//Cyl tags

OP160_HMI_MOVREM_Home_PB:BOOL;
OP160_HMI_MOVREM_Work_PB:BOOL;

OP160_HMI_Cycle_Start:					BOOL;
OP160_HMI_Reset:						BOOL;
OP160_HMI_Homing:						BOOL;
SR130_LH_Vert_Servo_Max_Lim:					BOOL;
SR130_RH_Vert_Servo_Max_Lim:					BOOL;
SR130_Clm_Vert_Max_Lim:					BOOL;


//Error

OP160_ErrorWord_0:    							 DINT;
OP160_ErrorWord_1:								 DINT;
OP160_ErrorWord_2:								 DINT;



//Robo bits

OP160_QC_Pick_Completed                            :BOOL;
OP160_Moverpresent                                 :BOOL;
OP160_PartPicked                                   :BOOL;
OP160_AutoPlaceSeq                                 :INT;
OP160_Robo_ProgramReset                            :BOOL;
OP160_Part_Placed                                  :BOOL;
OP160_MoverinStation                               :BOOL;
op160_place_both_component_ok                      :BOOL;
op160_place_1_ok_1_nok                             :BOOL;
op160_go_to_place                                  :BOOL;
op160_place_both_component_rej                     :BOOL;
op160_comp_Lh_ok_to_rbt                            :BOOL;
op160_comp_Lh_nok_to_rbt                           :BOOL;
op160_comp_rh_ok_to_rbt                            :BOOL;
op160_comp_rh_nok_to_rbt                           :BOOL;

END_VAR

VAR_GLOBAL PERSISTENT
	
Componenets_Produced        : DINT;
sampling_quantity           : INT;
sampling_request_qty        : INT;
sampling_request            : BOOL;
sampling_interval           : INT;

END_VAR

// ---- POUs/Programs/OP160/OP160_IO_Tag_Link.TcGVL

VAR_GLOBAL
	
	//Robo BYte Mapping Inputs
	OP160_Robo_IN_Byte1: BYTE_AS_BIT;
OP160_Robo_IN_6000_6007 AT %I*:BYTE;
OP160_Robo_IN_6008_6015 AT %I*:BYTE;
OP160_Robo_IN_6016_6023 AT %I*:BYTE;
OP160_Robo_IN_6024_6031 AT %I*:BYTE;
OP160_Robo_IN_6032_6039 AT %I*:BYTE;
OP160_Robo_IN_6040_6047 AT %I*:BYTE;
OP160_Robo_IN_6048_6055 AT %I*:BYTE;
OP160_Robo_IN_6056_6063 AT %I*:BYTE;
OP160_Robo_IN_6064_6071 AT %I*:BYTE;

//Robo Byte Mapping Out
OP160_Robo_Out_6000_6007 AT%Q*:BYTE;
OP160_Robo_Out_6008_6015 AT%Q*:BYTE;
OP160_Robo_Out_6016_6023 AT%Q*:BYTE;
OP160_Robo_Out_6024_6031 AT%Q*:BYTE;
OP160_Robo_Out_6032_6039 AT%Q*:BYTE;
OP160_Robo_Out_6040_6047 AT%Q*:BYTE;
OP160_Robo_Out_6048_6055 AT%Q*:BYTE;
OP160_Robo_Out_6056_6063 AT%Q*:BYTE;
OP160_Robo_Out_6064_6071 AT%Q*:BYTE;

	
	
//Robot Inputs
OP160_SO_Mirror_Auto_enable AT %I*:BOOL;
OP160_SO_Program_Execute AT %I*:BOOL;
OP160_SO_Program_Waiting AT %I*:BOOL;
OP160_SO_Program_Waiting2 AT %I*:BOOL;
OP160_SO_Stop_Status AT %I*:BOOL;
OP160_SO_Program_Sel_enabled_OP AT %I*:BOOL;
OP160_SO_During_error AT %I*:BOOL;
OP160_SO_During_Cycle_Stop AT %I*:BOOL;
OP160_SO_Mirror_SRVO_Off AT %I*:BOOL;
OP160_SO_Servo_ON_OFF_Status AT %I*:BOOL;
OP160_SO_Auto_Operation_Enable AT %I*:BOOL;
OP160_SO_Moving_Home AT %I*:BOOL;
OP160_SO_Spare1 AT %I*:BOOL;
OP160_SO_During_Machine_Lock AT %I*:BOOL;
OP160_SO_H_Error AT %I*:BOOL;
OP160_SO_L_Error AT %I*:BOOL;
OP160_SO_Caution AT %I*:BOOL;
OP160_SO_During_EMG_Stop AT %I*:BOOL;
OP160_SO_Teach_Mode AT %I*:BOOL;
OP160_SO_Auto_OP_Mode AT %I*:BOOL;
OP160_SO_Auto_Ext_Mode AT %I*:BOOL;
OP160_SO_TP_Enable AT %I*:BOOL;
OP160_SO_Heartbeat AT %I*:BOOL;
OP160_SO_Spare2 AT %I*:BOOL;
OP160_SO_Rbt_In_Home AT %I*:BOOL;
OP160_SO_Rbt_In_Pick_Zone AT %I*:BOOL;
OP160_SO_Rbt_In_Place_Zone AT %I*:BOOL;
OP160_SO_Rbt_In_Reject_Zone AT %I*:BOOL;
OP160_SO_Rbt_In_ATC_Zone AT %I*:BOOL;
OP160_SO_Spare4 AT %I*:BOOL;
OP160_SO_Spare5 AT %I*:BOOL;
OP160_SO_Spare6 AT %I*:BOOL;

OP160_GO_Mode_Ack AT %I*:BYTE;
OP160_GO_Variant_number_Ack AT %I*:BYTE;
OP160_GO_Position_Rchd_Ack AT %I*:BYTE;
OP160_GO_Auto_Status AT %I*:BYTE;
OP160_GO_Byte_Spare1 AT %I*:BYTE;
OP160_GO_Byte_Spare2 AT %I*:BYTE;
OP160_GO_Byte_Spare3 AT %I*:BYTE;
OP160_GO_Byte_Spare4 AT %I*:BYTE;
OP160_GO_Error_Number AT %I*:BYTE;
OP160_GO_Word_Spare AT %I*:BYTE;


OP160_EO_Sequence_Running AT %I*:BOOL;
OP160_EO_Sequence_Completed AT %I*:BOOL;
OP160_EO_Spring_Pick_Completed AT %I*:BOOL;
OP160_EO_Spring_Place_Pos_Reached AT %I*:BOOL;
OP160_EO_Spring_Place_Completed AT %I*:BOOL;
OP160_EO_NOK_Part_Dropped AT %I*:BOOL;
OP160_EO_Spare2 AT %I*:BOOL;
OP160_EO_Spare3 AT %I*:BOOL;
OP160_EO_Spare4 AT %I*:BOOL;
OP160_EO_Spare5 AT %I*:BOOL;
OP160_EO_Spare6 AT %I*:BOOL;
OP160_EO_Spare7 AT %I*:BOOL;
OP160_EO_Spare8 AT %I*:BOOL;
OP160_EO_Spare9 AT %I*:BOOL;
OP160_EO_Step_Reached AT %I*:BOOL;
OP160_EO_Spare11 AT %I*:BOOL;
OP160_EO_RO_Gripper1_Open AT %I*:BOOL;
OP160_EO_RO_Gripper1_Close AT %I*:BOOL;
OP160_EO_RO_Gripper2_Open AT %I*:BOOL;
OP160_EO_RO_Gripper2_Close AT %I*:BOOL;
OP160_EO_RO_ATC_Open AT %I*:BOOL;
OP160_EO_RO_ATC_Close AT %I*:BOOL;
OP160_EO_RO_Spare18 AT %I*:BOOL;
OP160_EO_RO_Spare19 AT %I*:BOOL;
OP160_EO_RI_Gripper1_Open_FB AT %I*:BOOL;
OP160_EO_RI_Gripper1_Close_FB AT %I*:BOOL;
OP160_EO_RI_Gripper2_Open_FB AT %I*:BOOL;
OP160_EO_RI_Gripper2_Close_FB AT %I*:BOOL;
OP160_EO_RI_ATC_Open_FB AT %I*:BOOL;
OP160_EO_RI_ATC_Close_FB AT %I*:BOOL;
OP160_EO_ATC_Tool_Presence_1 AT %I*:BOOL;
OP160_EO_ATC_Tool_Presence_2 AT %I*:BOOL;

//Robo Outputs
OP160_SI_Auto_Enable AT %Q*:BOOL;
OP160_SI_Start AT %Q*:BOOL;
OP160_SI_Stop AT %Q*:BOOL;
OP160_SI_Stop2 AT %Q*:BOOL;
OP160_SI_Spare1 AT %Q*:BOOL;
OP160_SI_Program_Reset AT %Q*:BOOL;
OP160_SI_Error_Reset AT %Q*:BOOL;
OP160_SI_Cycle_Stop AT %Q*:BOOL;
OP160_SI_Servo_OFF AT %Q*:BOOL;
OP160_SI_Servo_ON AT %Q*:BOOL;
OP160_SI_Operation_Enable AT %Q*:BOOL;
OP160_SI_Move_Home AT %Q*:BOOL;
OP160_SI_General_Output_reset AT %Q*:BOOL;
OP160_SI_Machine_Lock AT %Q*:BOOL;
OP160_SI_Spare2 AT %Q*:BOOL;
OP160_SI_Spare3 AT %Q*:BOOL;
OP160_SI_Spare4 AT %Q*:BOOL;
OP160_SI_Spare5 AT %Q*:BOOL;
OP160_SI_Spare6 AT %Q*:BOOL;
OP160_SI_Spare7 AT %Q*:BOOL;
OP160_SI_Spare8 AT %Q*:BOOL;
OP160_SI_Spare9 AT %Q*:BOOL;
OP160_SI_PLC_Heartbeat AT %Q*:BOOL;
OP160_SI_Dry_Run AT %Q*:BOOL;
OP160_SI_Homing_Start AT %Q*:BOOL;
OP160_SI_Pick_Zone_Safe AT %Q*:BOOL;
OP160_SI_Place_Zone_Safe AT %Q*:BOOL;
OP160_SI_Reject_Zone_Safe AT %Q*:BOOL;
OP160_SI_ATC_Tool_Safe AT %Q*:BOOL;
OP160_SI_Spare11 AT %Q*:BOOL;
OP160_SI_Spare12  AT %Q*:BOOL;
OP160_SI_Spare13 AT %Q*:BOOL;


OP160_GI_Mode AT %Q*:BYTE;
OP160_GI_Variant_number AT %Q*:BYTE;
OP160_GI_Position_Number AT %Q*:BYTE;
OP160_GI_Byte_Spare1 AT %Q*:BYTE;
OP160_GI_Byte_Spare2  AT %Q*:BYTE;
OP160_GI_Byte_Spare3 AT %Q*:BYTE;
OP160_GI_Byte_Spare4 AT %Q*:BYTE;
OP160_GI_Byte_Spare5 AT %Q*:BYTE;
OP160_GI_Word_Spare AT %Q*:BYTE;
OP160_GI_Word_Spare1 AT %Q*:BYTE;

OP160_EI_Manual_Seq_Start AT%Q*:BOOL;
OP160_EI_Spare2 AT%Q*:BOOL;
OP160_EI_Rdy_Pick_Spring AT%Q*:BOOL;
OP160_EI_Rdy_Place_Spring AT%Q*:BOOL;
OP160_EI_Insertion_Complete AT%Q*:BOOL;
OP160_EI_Rdy_Place_Rejection AT%Q*:BOOL;
OP160_EI_Spare4 AT%Q*:BOOL;
OP160_EI_Spare5 AT%Q*:BOOL;
OP160_EI_Spare6 AT%Q*:BOOL;
OP160_EI_Spare7 AT%Q*:BOOL;
OP160_EI_Spare8 AT%Q*:BOOL;
OP160_EI_Spare9 AT%Q*:BOOL;
OP160_EI_Spare10 AT%Q*:BOOL;
OP160_EI_Spare11 AT%Q*:BOOL;
OP160_EI_Step_Continue AT%Q*:BOOL;
OP160_EI_Spare13 AT%Q*:BOOL;
OP160_EI_Gripper1_Open AT%Q*:BOOL;
OP160_EI_Gripper1_Close AT%Q*:BOOL;
OP160_EI_Gripper2_Open AT%Q*:BOOL;
OP160_EI_Gripper2_Close AT%Q*:BOOL;
OP160_EI_ATC_Open AT%Q*:BOOL;
OP160_EI_ATC_Close AT%Q*:BOOL;
OP160_EI_Spare21 AT%Q*:BOOL;
OP160_EI_Spare22 AT%Q*:BOOL;
OP160_EI_Spare23 AT%Q*:BOOL;
OP160_EI_Spare24 AT%Q*:BOOL;
OP160_EI_Spare25 AT%Q*:BOOL;
OP160_EI_Spare26 AT%Q*:BOOL;
OP160_EI_Spare27 AT%Q*:BOOL;
OP160_EI_Spare28 AT%Q*:BOOL;
OP160_EI_Spare29 AT%Q*:BOOL;
OP160_EI_Spare30 AT%Q*:BOOL;


//Registerin
OP160_Robo_In6001 AT%I*:UINT;
OP160_Robo_In6002 AT%I*:UINT;
OP160_Robo_In6003 AT%I*:UINT;
OP160_Robo_In6004 AT%I*:UINT;
OP160_Robo_In6005 AT%I*:UINT;
OP160_Robo_In6006 AT%I*:UINT;
OP160_Robo_In6007 AT%I*:UINT;
OP160_Robo_In6008 AT%I*:UINT;
OP160_Robo_In6009 AT%I*:UINT;
OP160_Robo_In6010 AT%I*:UINT;
OP160_Robo_In6011 AT%I*:UINT;
OP160_Robo_In6012 AT%I*:UINT;

OP160_Robo_Out6001 AT%Q*:UINT;
OP160_Robo_Out6002 AT%Q*:UINT;
OP160_Robo_Out6003 AT%Q*:UINT;
OP160_Robo_Out6004 AT%Q*:UINT;
OP160_Robo_Out6005 AT%Q*:UINT;
OP160_Robo_Out6006 AT%Q*:UINT;
OP160_Robo_Out6007 AT%Q*:UINT;
OP160_Robo_Out6008 AT%Q*:UINT;
OP160_Robo_Out6009 AT%Q*:UINT;
OP160_Robo_Out6010 AT%Q*:UINT;


	OP160_SI_Insert_Cylinder_Home  : BOOL;
	OP160_SI_Spare10: BOOL;
	OP160_EI_Rdy_Pick_QC: BOOL;
	OP160_EI_Camera_OK: BOOL;
	OP160_EI_Camera_NOK: BOOL;
	OP160_EI_Rdy_Place_QC: BOOL;
	OP160_EI_Rdy_Place_Sample: BOOL;
	OP160_EI_Rdy_Place_Reject: BOOL;
	OP160_EI_Request_Changeover: BOOL;
	OP160_EI_Ready_To_Pick_Fixture: BOOL;
	OP160_EO_QC_Pick_Completed: BOOL;
	OP160_SO_Rbt_In_Change_Zone: BOOL;
	OP160_SO_Rbt_In_ATC: BOOL;
	OP160_EO_Camera_Trigger: BOOL;
	OP160_EO_Spare1: BOOL;
	OP160_EO_QC_Place_Completed: BOOL;
	OP160_EO_Sample_Place_Completed: BOOL;
	OP160_EO_Rejection_Place_Completed: BOOL;
	OP160_EO_Changeover_Running: BOOL;
	OP160_EO_Changeover_Completed: BOOL;
END_VAR

// ---- POUs/Programs/OP20/OP20_GVL.TcGVL

VAR_GLOBAL
//GENERAL
OP20_Auto:					BOOL;
OP20_Mode_Ack:				BOOL;
OP20_HomeRunning:			BOOL;
OP20_ErrorActive:			BOOL;
OP20_Home_PB:				BOOL;
OP20_Work_PB:				BOOL;
OP20_ManualSafetyBypass:	BOOL;
OP20_LightCurtainBypass:	BOOL;
OP20_OperationCompleted:	BOOL;
OP20_LampCheck:				BOOL;
OP20_MachineLamp:			BOOL;
OP20_ComponentOk:			BOOL;
OP20_ComponentNok:			BOOL;
OP20_RepeatBit:				BOOL;
OP20_HomingResetBit:		BOOL;
OP20_ControlledByRobo:		BOOL;
OP20_Any_Bypass:			BOOL;
OP20_ManualModeStatus:		INT;
OP20_ManualModeWord:		INT;
OP20_AutoRunning:			BOOL;
OP20_StepRunning:			BOOL;
OP20_StartEnable:   		BOOL;
OP20_HomeConditionOK:		BOOL;
OP20_Temp_hmeOK:			BOOL;
OP20_Machine_Stop: 			BOOL;
OP20_AutoSeq:				INT;
OP20_LH_AutoSeq: 			INT;
OP20_RH_AutoSeq: 			INT;
OP20_Homing_Seq:			INT;
OP20_Safety_OK:				BOOL;
OP20_Stop_Request: BOOL;

Automatic_Run:				BOOL;    //from master mode block
Manual_mode: 				BOOL;    //from master mode block

OP20_Prev_Stat_Operation_Completed: BOOL;
OP20_Prev_Comp_Status: INT;
OP20_Prev_LH_COMP_OK:BOOL;
OP20_Prev_LH_COMP_NOK:BOOL;
OP20_Prev_RH_COMP_OK:BOOL;
OP20_Prev_RH_COMP_NOK:BOOL;
OP20_LH_Operation_Completed:BOOL;
OP20_RH_Operation_Completed:BOOL;

temp_oil : BOOL;
//Servo controls
	OP20_Servo_Enable	: BOOL;
	OP20_Servo_Reset	: BOOL;
	SR20_Vert_servo: FB_Axis;
	SR20_Vert_servo_ctrl:Servo_Control;
	SR20_Vert_servo_status:stManualModeAxis;
//ModeSelection Outputs
//OP130_AutoSelected:		    BOOL;
OP20_ManualSelected:		BOOL;
OP20_StepSelected:			BOOL;
OP20_AutoSelected:		    BOOL;


//HMI Tags(From HMI)
OP20_HMI_AutoMode:						BOOL;
OP20_HMI_ManualMode:					BOOL;
OP20_HMI_StepMode:						BOOL;
OP20_HMI_CycleStart:					BOOL;
OP20_HMI_Reset:						    BOOL;
OP20_HMI_Homing:						BOOL;

OP20_HMI_Jog_Pos: BOOL;
OP20_HMI_Jog_Neg: BOOL;


OP20_AUTO_STP_NO: INT;

// MANUAL
		
// AUTO	

	OP20_FIXTURE_2					: INT;               //For the comp status in the fixture
	OP20_FIXTURE_1					: INT; 				 //For the comp status in the fixture
// SERVO VARIABLE
	OP20_VERT_SERVO_STRT			: BOOL;				// SERVO MOVE TO TARGET POSITION
	OP20_SERVO_POS_DONE				: BOOL;				// SERVO POSITION REACHED
	OP20_SERVO_ON_SFE_WRK			: BOOL;				// SERVO ACTUAL POSITION = SERVO SAFE POSITION
	OP20_SERVO_ON_WRK				: BOOL;				// SERVO ACTUAL POSITION = SERVO WORK POSITION
	OP20_SERVO_ON_HOME				: BOOL;				// SERVO ACTUAL POSITION = SERVO HOME POSITION	
	
	OP20_VERT_SERVO_HME_POS			: REAL := 0;         // SERVO IN HOME POSITION
	OP20_VERT_SERVO_POSITION		: LREAL ;			// SERVO ACTUAL POSITION
	OP20_VERT_SERVO_SFE_WRK_POS		: REAL := 0;		// SERVO SAFE WORK POSITION FROM RECEIPE
	OP20_VERT_SERVO_WRK_POS			: REAL := 40;		// SERVO WORK POSITION FROM RECEIPE	
	OP20_VERT_SERVO_TARGET			: REAL;				// SERVO AUTO TARGET POSITION

END_VAR

VAR_GLOBAL PERSISTENT
	
// MANUAL
	OP20_STN_ENABLE			: BOOL;				// FROM MASTER CONTROL BLOCK
	OP20_STN_RUNNING		: BOOL;
// AUTO
	OP20_BYPASS				: BOOL;				// OP20 ON-BYPASS / OFF-NOT BYPASSED
	OP20_LH_OIL_OK			: BOOL;				// TO MASTER CONTROL BLOCK OILLING LH OK BIT
	OP20_LH_OIL_NOK			: BOOL;				// TO MASTER CONTROL BLOCK OILLING LH NOK BIT
	OP20_RH_OIL_OK			: BOOL;				// TO MASTER CONTROL BLOCK OILLING RH OK BIT
	OP20_RH_OIL_NOK			: BOOL;				// TO MASTER CONTROL BLOCK OILLING RH NOK BIT
	
	OP20_OIL_TIMER			: INT:=100;			    	// AUTO DELAY TIMER AFTER SERVO REACH WORK
	OP20_Cycle_time			: UDINT;
//Setting Parameters
    OP20_HMI_Servo_Speed      : REAL;
    OP20_HMI_Low_Limit		 : REAL;
    OP20_HMI_High_Limit		 : REAL;
	OP20_HMI_Safe_Home		 : REAL;
	OP20_HMI_Safe_Work		 : REAL;
//Error
	OP20_ErrorWord_0: DINT;
	OP20_ErrorWord_1: DINT;
	OP20_ErrorWord_2: DINT;
	
		Oil_Region : REAL:=6;
END_VAR

VAR_GLOBAL 
	temp:BOOL;
END_VAR

// ---- POUs/Programs/OP20/OP20_Recipe.TcGVL

VAR_GLOBAL PERSISTENT
	OP20_DLY_OIL_ON : INT;
	OP20_VERT_SERVO_WORK_POS : REAL;
	OP20_VERT_SERVO_SFE_WORK_POS : REAL;	
END_VAR

// ---- POUs/Programs/OP30/OP30_GVL.TcGVL

VAR_GLOBAL
			
//GENERAL
OP30_Auto:					BOOL;
OP30_Mode_Ack:				BOOL;
OP30_HomeRunning:			BOOL;
OP30_ErrorActive:			BOOL;
OP30_Home_PB:				BOOL;
OP30_Work_PB:				BOOL;
OP30_ManualSafetyBypass:	BOOL;
OP30_LightCurtainBypass:	BOOL;
OP30_OperationCompleted:	BOOL;
OP30_LampCheck:				BOOL;
OP30_MachineLamp:			BOOL;
OP30_ComponentOk:			BOOL;
OP30_ComponentNok:			BOOL;
OP30_RepeatBit:				BOOL;
OP30_HomingResetBit:		BOOL;
OP30_ControlledByRobo:		BOOL;
OP30_Any_Bypass:			BOOL;
OP30_ManualModeStatus:		INT;
OP30_ManualModeWord:		INT;
OP30_AutoRunning:			BOOL;
OP30_StepRunning:			BOOL;
OP30_StartEnable:   		BOOL;
OP30_HomeConditionOK:		BOOL;
OP30_Temp_hmeOK:			BOOL;
OP30_Machine_Stop: 			BOOL;
OP30_AutoSeq:				INT;
OP30_LH_AutoSeq: 			INT;
OP30_RH_AutoSeq: 			INT;
OP30_Homing_Seq:			INT;
OP30_Safety_OK:				BOOL;
OP30_STN_ENABLE				: BOOL;
OP30_Stop_Request			: BOOL;
OP30_Conveyor_ON			: BOOL;
	
OP30_ManualSelected:		BOOL;
OP30_StepSelected:			BOOL;
OP30_AutoSelected:		    BOOL;

OP30_HMI_AutoMode:						BOOL;
OP30_HMI_ManualMode:					BOOL;
OP30_HMI_StepMode:						BOOL;
OP30_HMI_CycleStart:					BOOL;
OP30_HMI_Cycle_Start:					BOOL;
OP30_HMI_Reset:						    BOOL;
OP30_HMI_Homing:						BOOL;

SR30_Vert_servo: FB_Axis;
SR30_Vert_servo_ctrl:Servo_Control;
SR30_Vert_servo_status:stManualModeAxis;

SR30_Hori_servo: FB_Axis;


SR30_Conv_servo: FB_Axis;
SR30_Conv_servo_ctrl:Servo_Control;
SR30_Conv_servo_status:stManualModeAxis;

OP30_Gripper_LH : FB_Schunk;
OP30_Gripper_LH_Manual_Axis: stManualModeAxis; 
OP30_Gripper_LH_Gripper_ctrl: Servo_Control; 

OP30_GIUDE_GRP: FB_Axis_FESTO;


OP30_Gripper_Current     : REAL;
OP30_Gripper_Acceleration: REAL;
OP30_Gripper_Jerk        : REAL;

OP30_Gripper_RH : FB_Schunk;
OP30_Gripper_RH_Manual_Axis: stManualModeAxis;
OP30_Gripper_RH_Gripper_ctrl: Servo_Control; 

OP30_Drum_feeder_ON 	  : BOOL;
OP30_Drum_feeder_State : BOOL;

Camera_LH_Trig : BOOL;
Camera_LH_OK   : BOOL;

Camera_RH_Trig : BOOL;
Camera_RH_OK   : BOOL;

//Cylinder
CR30_LH_Rej_Cyl: Cylinder_Block;
CR30_RH_Rej_Cyl: Cylinder_Block;
CR30_LH_Rej_Cyl_status : INT;
CR30_RH_Rej_Cyl_status : INT;
OP30_HMI_LH_Rej_Cyl_Home_PB : BOOL;
OP30_HMI_LH_Rej_Cyl_Work_PB : BOOL;
OP30_HMI_RH_Rej_Cyl_Home_PB : BOOL;
OP30_HMI_RH_Rej_Cyl_Work_PB : BOOL;

//conveyor
OP30_pick_ready     : BOOL;
OP30_pick_done      : BOOL;
OP30_Conv_Fwd_Time	: INT;
OP30_Conv_Rev_Time	: INT;
OP30_Conveyor_FWD_Speed	: REAL;
OP30_Conveyor_REV_Speed	: REAL;

//
CR30_LH_Rej_Cyl_wrk  : BOOL;
CR30_LH_Rej_Cyl_hme  : BOOL;
CR30_RH_Rej_Cyl_wrk  : BOOL;
CR30_RH_Rej_Cyl_hme  : BOOL;


//Schunk Gripper
HwIn1 	 	AT%I*:	ARRAY [0..8] OF WORD;
HwIn2  		AT%I*:	ARRAY [0..8] OF WORD;
HwIn3 	 	AT%I*:	ARRAY [0..8] OF WORD;
HwIn4  		AT%I*:	ARRAY [0..8] OF WORD;
                    
HwOut1		AT%Q*:	ARRAY [0..11] OF WORD;
HwOut2		AT%Q*:	ARRAY [0..11] OF WORD;
HwOut3		AT%Q*:	ARRAY [0..11] OF WORD;
HwOut4		AT%Q*:	ARRAY [0..11] OF WORD;

//Camera
	OP30_Camera_Trigger				  : BOOL;
	OP30_LH_Clr_OK					  : BOOL;
	OP30_LH_Clr_NOK					  : BOOL;
	OP30_LH_Size_OK					  : BOOL;
	OP30_LH_Size_NOK				  : BOOL;
	OP30_LH_Part_OK					  : BOOL;
	OP30_LH_Part_NOK				  : BOOL;
	OP30_Size_Rej					  : BOOL;
	OP30_Size_Rej_Complete			  : BOOL;
	OP30_One_Cycle				      : BOOL;
	OP30_LH_Camera_OK 				  : BOOL;
	OP30_LH_Camera_NOK                : BOOL;
	OP30_RH_Camera_OK                 : BOOL;
	OP30_RH_Camera_NOK                : BOOL;
	OP30_Camera_Done				  : BOOL;
	
	OP30_RH_Clr_OK					  : BOOL;
	OP30_RH_Clr_NOK					  : BOOL;
	OP30_RH_Size_OK					  : BOOL;
	OP30_RH_Size_NOK				  : BOOL;
	OP30_RH_Part_OK					  : BOOL;
	OP30_RH_Part_NOK				  : BOOL;	
	
	OP30_LH_Camera_Trigger		      : BOOL;
	OP30_LH_Camera_Job_Change_start   : BOOL;
	OP30_LH_Camera_Error			  : BOOL;
	OP30_LH_Camera_Ready			  : BOOL;
	OP30_LH_Camera_Online			  : BOOL;	
	OP30_LH_Job_Change_Complete		    : BOOL;
	OP30_LH_Job_Change_Error   		    : BOOL;
	OP30_LH_Picture_Taken      		    : BOOL;	
	OP30_LH_Error_status			    : STRING;
	OP30_LH_Target_Job_ID				: UINT;
	OP30_LH_Loaded_Job_ID		    	: UINT;
	
	OP30_RH_Camera_Trigger		      : BOOL;
	OP30_RH_Camera_Job_Change_start   : BOOL;
	OP30_RH_Camera_Error			  : BOOL;
	OP30_RH_Camera_Ready			  : BOOL;
	OP30_RH_Camera_Online			  : BOOL;
	OP30_RH_Job_Change_Complete		    : BOOL;
	OP30_RH_Job_Change_Error   		    : BOOL;
	OP30_RH_Picture_Taken      		    : BOOL;
	OP30_RH_Error_status				: STRING;
	OP30_RH_Target_Job_ID				: UINT;
	OP30_RH_Loaded_Job_ID		    	: UINT;	

END_VAR

VAR_GLOBAL PERSISTENT
	
	

	OP30_Cycle_time : UDINT;
	
	OP30_Gripper_LH_Open  : BOOL;
    OP30_Gripper_LH_Close : BOOL;
    OP30_Gripper_LH_State : BOOL;  //1-- Open 0--Close
    
    OP30_Gripper_RH_Open  : BOOL;
    OP30_Gripper_RH_Close : BOOL;
    OP30_Gripper_RH_State : BOOL;


    OP30_VERT_SERVO_POS_DONE	    	: BOOL;
    OP30_VERT_SERVO_ON_SFE_WRK			: BOOL;
    OP30_VERT_SERVO_ON_WRK_PICK			: BOOL;
	OP30_VERT_SERVO_ON_WRK_PLACE		: BOOL;
    OP30_VERT_SERVO_ON_HOME				: BOOL;
	  
	OP30_VERT_SERVO_POSITION		: LREAL ;
	OP30_VERT_SERVO_HME_POS			: REAL := 0;  				
	OP30_VERT_SERVO_SFE_WRK_POS		: REAL := 10;		
	OP30_VERT_SERVO_PICK_POS		: REAL := 64;	
	OP30_VERT_SERVO_PLACE_POS		: REAL := 80;

    OP30_HORI_SERVO_POS_DONE	    	: BOOL;
    OP30_HORI_SERVO_ON_SFE_WRK			: BOOL;
    OP30_HORI_SERVO_ON_WRK_PICK			: BOOL;
    OP30_HORI_SERVO_ON_SFE_WRK_PICK		: BOOL;	
	OP30_HORI_SERVO_ON_WRK_PLACE		: BOOL;
    OP30_HORI_SERVO_ON_HOME				: BOOL;
	  
	OP30_HORI_SERVO_POSITION		: LREAL ;
	OP30_HORI_SERVO_HME_POS			: REAL := -40;  				
	OP30_HORI_SERVO_SFE_WRK_POS		: REAL :=-40;
	OP30_HORI_SERVO_SAFE_PICK_POS	: REAL := 100; 		
	OP30_HORI_SERVO_PICK_POS		: REAL :=149.8;	
	OP30_HORI_SERVO_PLACE_POS		: REAL :=36.6;
	
    OP30_CONV_SERVO_POS_DONE	    	: BOOL;
    OP30_CONV_SERVO_ON_SFE_WRK			: BOOL;
    OP30_CONV_SERVO_ON_WRK				: BOOL;
    OP30_CONV_SERVO_ON_HOME				: BOOL;
	
	OP30_CONV_SERVO_POSITION		: LREAL ;
	OP30_CONV_SERVO_HME_POS			: REAL; 				
	OP30_CONV_SERVO_SFE_WRK_POS		: REAL ;		
	OP30_CONV_SERVO_WRK_POS			: REAL;
	
//Drum_Feeder
	OP30_Drum_Feed_Motor_Speed		AT %Q*  : INT;	
	OP30_HMI_Drum_Feed_Mtr_Speed_IP		: INT;
	OP30_Drum_Feed_Mtr_Speed_Select		: BOOL;
	OP30_Drum_Feed_Mtr_Run_Fwd 			: BOOL;
	OP30_Drum_Feed_Mtr_Reset   			: BOOL;
//Error
OP30_ErrorWord_0: DINT;
OP30_ErrorWord_1: DINT;
OP30_ErrorWord_2: DINT;	

//Setting Parameters
    OP30_HMI_Servo_Speed_Vertical     : REAL ;
	OP30_HMI_Servo_Speed_Horizontal	  : REAL ;
    OP30_HMI_Hori_Low_Limit		 : REAL:=0;
    OP30_HMI_Hori_High_Limit     : REAL:=200;
    OP30_HMI_Vert_Low_Limit		 : REAL:=0;
    OP30_HMI_Vert_High_Limit     : REAL:=100;	

	OP30_Vert_Ser_Safe_Pos			: REAL;
	OP30_Hori_Ser_Rej_Pos			: REAL;	
	OP30_Hori_Ser_Jerk_Pos			: REAL :=1;		
	OP30_Drum_Freq		  			: REAL;
	
	OP30_Conv_Fwd_Time_6_3			: INT:=750;
	OP30_Conv_Fwd_Speed_6_3			: INT:=150;
	OP30_Conv_Rev_Time_6_3			: INT:=500;
	OP30_Conv_Rev_Speed_6_3			: INT:=-100;
	
	OP30_Conv_Fwd_Pos				: REAL :=10;
	OP30_Conv_Rev_Pos				: REAL  :=5;

	OP30_Conv_Fwd_Time_7_89			: INT:=750;
	OP30_Conv_Fwd_Speed_7_89		: INT:=150;
	OP30_Conv_Rev_Time_7_89			: INT:=500;
	OP30_Conv_Rev_Speed_7_89		: INT:=-100;		
	
	OP30_Conveyor_Speed				: REAL;
	OP30_Model						: STRING[80];
	OP30_Gripper_WRK_POS			: REAL :=2;
	
	OP30_Grip_LH_Bypass				: BOOL;
	OP30_Grip_RH_Bypass				: BOOL;
	OP30_Guide_Pos					: REAL :=75;
	
//Drum Timers
	OP30_Drum_ON_Time				: INT :=4000;
	OP30_Drum_OFF_Time				: INT :=1000;
	
END_VAR

// ---- POUs/Programs/OP30/OP30_HMI_TAGS.TcGVL
VAR_GLOBAL
	
OP30_GIUDE_GRP_Manual_Axis: stManualModeAxis; 
OP30_GIUDE_GRP_ctrl: Servo_Control;	

SR30_Hori_servo_ctrl:Servo_Control;
SR30_Hori_servo_status:stManualModeAxis;

END_VAR

// ---- POUs/Programs/OP30/OP30_Recipe.TcGVL

VAR_GLOBAL
END_VAR

// ---- POUs/Programs/OP40/OP40_GVL.TcGVL
VAR_GLOBAL
	
